C03599=1028.840,190.655,-111.620,169.303,45.603,158.612
C03600=1028.846,190.904,-111.645,169.306,45.600,158.612
C03601=1028.852,191.152,-111.668,169.310,45.598,158.612
C03602=1028.858,191.400,-111.692,169.315,45.595,158.612
C03603=1028.864,191.650,-111.717,169.318,45.592,158.612
C03604=1028.870,191.898,-111.740,169.321,45.590,158.612
C03605=1028.876,192.147,-111.765,169.325,45.587,158.612
C03606=1028.881,192.396,-111.788,169.328,45.585,158.611
C03607=1028.887,192.645,-111.812,169.332,45.583,158.611
C03608=1028.893,192.894,-111.836,169.335,45.580,158.611
C03609=1028.899,193.142,-111.860,169.338,45.578,158.611
C03610=1028.905,193.391,-111.884,169.343,45.575,158.611
C03611=1028.911,193.640,-111.908,169.346,45.572,158.611
C03612=1028.917,193.889,-111.933,169.350,45.570,158.611
C03613=1028.923,194.137,-111.956,169.353,45.567,158.610
C03614=1028.929,194.386,-111.981,169.357,45.565,158.610
C03615=1028.935,194.635,-112.005,169.360,45.563,158.610
C03616=1028.941,194.884,-112.029,169.364,45.560,158.610
C03617=1028.947,195.132,-112.053,169.368,45.557,158.610
C03618=1028.953,195.382,-112.078,169.372,45.555,158.610
C03619=1028.959,195.630,-112.101,169.375,45.552,158.610
C03620=1028.966,195.879,-112.125,169.378,45.550,158.610
C03621=1028.971,196.127,-112.149,169.383,45.547,158.609
C03622=1028.978,196.376,-112.173,169.386,45.545,158.609
C03623=1028.983,196.625,-112.198,169.390,45.542,158.609
C03624=1028.990,196.874,-112.222,169.393,45.540,158.609
C03625=1028.995,197.123,-112.246,169.396,45.537,158.609
C03626=1029.002,197.372,-112.270,169.401,45.535,158.609
C03627=1029.007,197.619,-112.295,169.404,45.532,158.609
C03628=1029.014,197.868,-112.319,169.408,45.530,158.609
C03629=1029.019,198.117,-112.343,169.411,45.528,158.609
C03630=1029.026,198.366,-112.367,169.416,45.525,158.609
C03631=1029.032,198.615,-112.392,169.419,45.522,158.608
C03632=1029.038,198.864,-112.416,169.423,45.520,158.608
C03633=1029.044,199.113,-112.440,169.426,45.518,158.608
C03634=1029.050,199.361,-112.465,169.431,45.515,158.608
C03635=1029.057,199.610,-112.489,169.434,45.512,158.608
C03636=1029.062,199.859,-112.513,169.438,45.510,158.608
C03637=1029.068,200.107,-112.537,169.441,45.507,158.608
C03638=1029.074,200.356,-112.562,169.445,45.505,158.608
C03639=1029.081,200.605,-112.587,169.449,45.503,158.607
C03640=1029.086,200.854,-112.611,169.452,45.500,158.607
C03641=1029.092,201.102,-112.636,169.456,45.498,158.607
C03642=1029.098,201.351,-112.660,169.460,45.496,158.607
C03643=1029.104,201.600,-112.685,169.464,45.494,158.607
C03644=1029.110,201.849,-112.710,169.468,45.491,158.607
C03645=1029.116,202.097,-112.734,169.471,45.488,158.607
C03646=1029.122,202.346,-112.760,169.474,45.486,158.607
C03647=1029.128,202.595,-112.784,169.479,45.484,158.607
C03648=1029.134,202.843,-112.809,169.482,45.482,158.607
C03649=1029.140,203.092,-112.833,169.486,45.479,158.607
C03650=1029.146,203.341,-112.858,169.490,45.477,158.606
C03651=1029.151,203.589,-112.883,169.494,45.475,158.606
C03652=1029.157,203.839,-112.908,169.498,45.472,158.606
C03653=1029.182,204.885,-113.012,169.864,45.576,158.667
C03654=1029.194,205.258,-113.051,169.867,45.574,158.667
C03655=1029.203,205.632,-113.091,169.872,45.571,158.667
C03656=1029.213,206.005,-113.130,169.876,45.569,158.667
C03657=1029.223,206.378,-113.169,169.880,45.566,158.667
C03658=1029.230,206.628,-113.195,169.883,45.565,158.667
C03659=1029.236,206.876,-113.221,169.886,45.564,158.667
C03660=1029.243,207.124,-113.248,169.889,45.562,158.667
C03661=1029.250,207.372,-113.274,169.892,45.560,158.667
C03662=1029.256,207.621,-113.301,169.895,45.559,158.667
C03663=1029.263,207.870,-113.327,169.897,45.557,158.667
C03664=1029.270,208.118,-113.353,169.900,45.556,158.667
C03665=1029.277,208.367,-113.380,169.903,45.554,158.667
C03666=1029.284,208.615,-113.406,169.905,45.553,158.667
C03667=1029.290,208.864,-113.433,169.908,45.551,158.667
C03668=1029.297,209.112,-113.459,169.911,45.550,158.667
C03669=1029.304,209.361,-113.485,169.914,45.549,158.667
C03670=1029.309,209.609,-113.512,169.916,45.547,158.666
C03671=1029.317,209.858,-113.538,169.919,45.545,158.666
C03672=1029.324,210.107,-113.565,169.923,45.544,158.666
C03673=1029.330,210.355,-113.591,169.926,45.542,158.666
C03674=1029.337,210.604,-113.618,169.928,45.541,158.667
C03675=1029.343,210.852,-113.644,169.931,45.540,158.667
C03676=1029.350,211.101,-113.670,169.934,45.538,158.666
C03677=1029.356,211.349,-113.697,169.936,45.536,158.666
C03678=1029.363,211.598,-113.723,169.939,45.535,158.666
C03679=1029.370,211.846,-113.751,169.942,45.534,158.666
C03680=1029.376,212.094,-113.777,169.945,45.532,158.666
C03681=1029.383,212.343,-113.804,169.948,45.531,158.666
C03682=1029.389,212.591,-113.830,169.950,45.530,158.666
C03683=1029.396,212.840,-113.856,169.954,45.528,158.666
C03684=1029.403,213.089,-113.883,169.957,45.527,158.667
C03685=1029.409,213.337,-113.910,169.960,45.525,158.667
C03686=1029.416,213.586,-113.937,169.962,45.524,158.667
C03687=1029.422,213.834,-113.963,169.965,45.523,158.667
C03688=1029.429,214.083,-113.990,169.968,45.521,158.667
C03689=1029.436,214.331,-114.017,169.970,45.519,158.666
C03690=1029.442,214.579,-114.044,169.973,45.518,158.666
C03691=1029.449,214.828,-114.071,169.976,45.517,158.666
C03692=1029.456,215.077,-114.097,169.979,45.515,158.666
C03693=1029.462,215.325,-114.124,169.983,45.514,158.666
C03694=1029.469,215.573,-114.151,169.985,45.512,158.666
C03695=1029.476,215.822,-114.178,169.988,45.511,158.667
C03696=1029.482,216.070,-114.204,169.991,45.510,158.667
C03697=1029.489,216.319,-114.232,169.994,45.508,158.667
C03698=1029.496,216.568,-114.258,169.996,45.507,158.667
C03699=1029.502,216.816,-114.285,169.999,45.506,158.667
C03700=1029.509,217.064,-114.312,170.002,45.504,158.667
C03701=1029.516,217.313,-114.339,170.006,45.503,158.667
C03702=1029.523,217.562,-114.365,170.009,45.501,158.667
C03703=1029.529,217.810,-114.393,170.011,45.500,158.667
C03704=1029.536,218.058,-114.419,170.014,45.499,158.667
C03705=1029.543,218.307,-114.447,170.017,45.497,158.667
C03706=1029.549,218.555,-114.473,170.020,45.496,158.667
C03707=1029.556,218.804,-114.499,170.023,45.495,158.667
C03708=1029.563,219.052,-114.527,170.026,45.493,158.667
C03709=1029.570,219.301,-114.553,170.029,45.492,158.667
C03710=1029.579,219.679,-114.594,170.034,45.490,158.667
C03711=1029.589,220.058,-114.636,170.037,45.488,158.667
C03712=1029.599,220.437,-114.678,170.042,45.486,158.667
C03713=1029.609,220.816,-114.719,170.047,45.484,158.667
C03714=1029.616,221.065,-114.746,170.050,45.483,158.667
C03715=1029.623,221.313,-114.773,170.052,45.482,158.667
C03716=1029.630,221.562,-114.800,170.055,45.480,158.667
C03717=1029.636,221.810,-114.828,170.058,45.479,158.667
C03718=1029.642,222.059,-114.855,170.062,45.477,158.667
C03719=1029.649,222.307,-114.882,170.064,45.476,158.667
C03720=1029.656,222.556,-114.910,170.068,45.475,158.667
C03721=1029.662,222.804,-114.936,170.070,45.474,158.667
C03722=1029.669,223.053,-114.964,170.073,45.473,158.667
C03723=1029.676,223.301,-114.991,170.076,45.471,158.667
C03724=1029.682,223.550,-115.018,170.079,45.470,158.667
C03725=1029.689,223.798,-115.046,170.082,45.468,158.667
C03726=1029.695,224.046,-115.073,170.085,45.467,158.667
C03727=1029.701,224.295,-115.100,170.088,45.466,158.668
C03728=1029.709,224.543,-115.127,170.091,45.465,158.668
C03729=1029.716,224.792,-115.155,170.094,45.464,158.668
C03730=1029.722,225.041,-115.182,170.098,45.462,158.668
C03731=1029.729,225.289,-115.210,170.100,45.461,158.668
C03732=1029.735,225.537,-115.237,170.103,45.460,158.668
C03733=1029.742,225.785,-115.264,170.106,45.459,158.668
C03734=1029.749,226.034,-115.291,170.109,45.457,158.668
C03735=1029.755,226.282,-115.319,170.112,45.456,158.668
C03736=1029.763,226.531,-115.346,170.115,45.454,158.668
C03737=1029.769,226.779,-115.374,170.118,45.454,158.668
C03738=1029.776,227.027,-115.402,170.121,45.452,158.668
C03739=1029.782,227.276,-115.428,170.124,45.451,158.668
C03740=1029.789,227.524,-115.455,170.127,45.450,158.668
C03741=1029.796,227.772,-115.483,170.131,45.448,158.668
C03742=1029.803,228.021,-115.511,170.134,45.447,158.668
C03743=1029.809,228.269,-115.539,170.136,45.446,158.668
C03744=1029.816,228.518,-115.566,170.139,45.445,158.668
C03745=1029.823,228.766,-115.594,170.142,45.444,158.669
C03746=1029.829,229.015,-115.622,170.146,45.443,158.669
C03747=1029.835,229.262,-115.649,170.149,45.441,158.669
C03748=1029.842,229.511,-115.676,170.152,45.440,158.669
C03749=1029.848,229.760,-115.704,170.155,45.439,158.669
C03750=1029.855,230.008,-115.732,170.157,45.438,158.669
C03751=1029.862,230.257,-115.759,170.161,45.437,158.669
C03752=1029.868,230.505,-115.787,170.164,45.436,158.669
C03753=1029.875,230.754,-115.815,170.167,45.434,158.669
C03754=1029.882,231.002,-115.843,170.170,45.433,158.669
C03755=1029.888,231.250,-115.870,170.173,45.432,158.669
C03756=1029.895,231.499,-115.899,170.176,45.431,158.669
C03757=1029.901,231.747,-115.927,170.180,45.430,158.669
C03758=1029.908,231.995,-115.955,170.182,45.429,158.669
C03759=1029.914,232.243,-115.982,170.185,45.428,158.670
C03760=1029.921,232.492,-116.010,170.188,45.427,158.670
C03761=1029.928,232.740,-116.038,170.191,45.426,158.670
C03762=1029.933,232.989,-116.066,170.195,45.424,158.670
C03763=1029.940,233.237,-116.094,170.198,45.424,158.670
C03764=1029.947,233.485,-116.122,170.201,45.422,158.670
C03765=1029.954,233.734,-116.150,170.204,45.422,158.670
C03766=1029.964,234.105,-116.192,170.209,45.420,158.670
C03767=1029.973,234.476,-116.234,170.213,45.418,158.670
C03768=1029.984,234.848,-116.275,170.218,45.416,158.671
C03769=1029.994,235.219,-116.317,170.223,45.414,158.671
C03770=1030.000,235.467,-116.345,170.226,45.414,158.671
C03771=1030.006,235.716,-116.373,170.229,45.412,158.671
C03772=1030.013,235.964,-116.401,170.232,45.412,158.671
C03773=1030.020,236.212,-116.429,170.236,45.410,158.671
C03774=1030.026,236.460,-116.457,170.239,45.409,158.671
C03775=1030.033,236.709,-116.485,170.241,45.408,158.671
C03776=1030.040,236.958,-116.513,170.244,45.407,158.671
C03777=1030.047,237.206,-116.542,170.248,45.406,158.671
C03778=1030.053,237.455,-116.570,170.251,45.405,158.672
C03779=1030.060,237.703,-116.597,170.254,45.404,158.672
C03780=1030.067,237.951,-116.626,170.257,45.403,158.672
C03781=1030.073,238.200,-116.654,170.261,45.401,158.672
C03782=1030.080,238.448,-116.682,170.264,45.401,158.672
C03783=1030.087,238.696,-116.710,170.267,45.400,158.672
C03784=1030.093,238.944,-116.738,170.270,45.399,158.672
C03785=1030.100,239.192,-116.767,170.274,45.398,158.672
C03786=1030.106,239.441,-116.795,170.277,45.396,158.672
C03787=1030.113,239.689,-116.823,170.280,45.396,158.673
C03788=1030.120,239.937,-116.851,170.282,45.394,158.673
C03789=1030.126,240.187,-116.880,170.286,45.394,158.673
C03790=1030.133,240.434,-116.908,170.289,45.393,158.673
C03791=1030.139,240.683,-116.936,170.292,45.392,158.673
C03792=1030.146,240.931,-116.965,170.295,45.391,158.673
C03793=1030.153,241.179,-116.993,170.299,45.390,158.673
C03794=1030.159,241.428,-117.022,170.302,45.389,158.673
C03795=1030.166,241.675,-117.050,170.305,45.388,158.674
C03796=1030.172,241.924,-117.078,170.309,45.387,158.674
C03797=1030.179,242.172,-117.107,170.312,45.386,158.674
C03798=1030.186,242.421,-117.136,170.315,45.385,158.674
C03799=1030.193,242.669,-117.164,170.318,45.384,158.674
C03800=1030.199,242.917,-117.193,170.322,45.383,158.674
C03801=1030.206,243.165,-117.222,170.325,45.382,158.674
C03802=1030.212,243.414,-117.250,170.328,45.381,158.675
C03803=1030.219,243.662,-117.278,170.331,45.381,158.675
C03804=1030.225,243.910,-117.307,170.335,45.380,158.675
C03805=1030.232,244.159,-117.335,170.338,45.378,158.675
C03806=1030.239,244.407,-117.364,170.341,45.378,158.675
C03807=1030.245,244.655,-117.394,170.345,45.377,158.675
C03808=1030.251,244.903,-117.423,170.348,45.376,158.675
C03809=1030.258,245.152,-117.450,170.351,45.375,158.676
C03810=1030.264,245.400,-117.479,170.354,45.375,158.676
C03811=1030.270,245.648,-117.508,170.358,45.373,158.676
C03812=1030.277,245.897,-117.538,170.361,45.372,158.676
C03813=1030.284,246.145,-117.566,170.364,45.372,158.676
C03814=1030.290,246.393,-117.595,170.367,45.371,158.676
C03815=1030.297,246.641,-117.624,170.371,45.370,158.677
C03816=1030.303,246.890,-117.653,170.374,45.369,158.677
C03817=1030.310,247.138,-117.681,170.377,45.369,158.677
C03818=1030.317,247.386,-117.710,170.380,45.368,158.677
C03819=1030.323,247.635,-117.740,170.384,45.367,158.677
C03820=1030.329,247.883,-117.769,170.387,45.366,158.677
C03821=1030.335,248.131,-117.798,170.390,45.365,158.678
C03822=1030.346,248.497,-117.840,170.395,45.364,158.678
C03823=1030.355,248.861,-117.883,170.400,45.363,158.678
C03824=1030.365,249.227,-117.926,170.405,45.362,158.678
C03825=1030.374,249.592,-117.968,170.410,45.360,158.679
C03826=1030.381,249.840,-117.997,170.413,45.360,158.679
C03827=1030.387,250.089,-118.027,170.416,45.359,158.679
C03828=1030.394,250.337,-118.055,170.420,45.358,158.679
C03829=1030.401,250.585,-118.084,170.423,45.357,158.679
C03830=1030.407,250.834,-118.113,170.426,45.357,158.680
C03831=1030.414,251.082,-118.142,170.430,45.356,158.680
C03832=1030.420,251.330,-118.172,170.433,45.355,158.680
C03833=1030.427,251.577,-118.201,170.436,45.354,158.680
C03834=1030.434,251.826,-118.230,170.440,45.353,158.680
C03835=1030.440,252.074,-118.259,170.443,45.353,158.680
C03836=1030.447,252.323,-118.288,170.446,45.352,158.681
C03837=1030.453,252.571,-118.318,170.451,45.351,158.681
C03838=1030.460,252.819,-118.346,170.454,45.350,158.681
C03839=1030.467,253.067,-118.375,170.457,45.349,158.681
C03840=1030.474,253.316,-118.405,170.461,45.349,158.681
C03841=1030.480,253.564,-118.434,170.464,45.348,158.682
C03842=1030.487,253.813,-118.464,170.468,45.347,158.682
C03843=1030.494,254.060,-118.492,170.471,45.347,158.682
C03844=1030.500,254.308,-118.521,170.474,45.346,158.682
C03845=1030.507,254.557,-118.551,170.478,45.345,158.682
C03846=1030.514,254.805,-118.580,170.481,45.344,158.682
C03847=1030.520,255.054,-118.610,170.485,45.343,158.683
C03848=1030.527,255.301,-118.638,170.488,45.343,158.683
C03849=1030.534,255.549,-118.668,170.491,45.342,158.683
C03850=1030.541,255.798,-118.697,170.495,45.341,158.683
C03851=1030.547,256.046,-118.726,170.498,45.340,158.683
C03852=1030.554,256.294,-118.756,170.502,45.339,158.684
C03853=1030.560,256.542,-118.785,170.505,45.339,158.684
C03854=1030.568,256.791,-118.814,170.508,45.338,158.684
C03855=1030.575,257.038,-118.844,170.512,45.337,158.684
C03856=1030.581,257.287,-118.873,170.515,45.336,158.684
C03857=1030.588,257.535,-118.903,170.519,45.335,158.685
C03858=1030.594,257.783,-118.932,170.522,45.335,158.685
C03859=1030.602,258.031,-118.961,170.525,45.334,158.685
C03860=1030.608,258.279,-118.990,170.529,45.333,158.685
C03861=1030.615,258.528,-119.020,170.533,45.333,158.685
C03862=1030.622,258.776,-119.049,170.537,45.332,158.686
C03863=1030.629,259.024,-119.079,170.540,45.331,158.686
C03864=1030.636,259.273,-119.109,170.544,45.331,158.686
C03865=1030.643,259.520,-119.138,170.547,45.330,158.686
C03866=1030.650,259.769,-119.167,170.551,45.329,158.686
C03867=1030.656,260.017,-119.196,170.554,45.328,158.687
C03868=1030.663,260.265,-119.227,170.558,45.327,158.687
C03869=1030.669,260.513,-119.256,170.561,45.327,158.687
C03870=1030.676,260.762,-119.286,170.564,45.327,158.687
C03871=1030.684,261.009,-119.315,170.568,45.326,158.688
C03872=1030.691,261.258,-119.344,170.571,45.325,158.688
C03873=1030.696,261.505,-119.375,170.575,45.324,158.688
C03874=1030.703,261.754,-119.404,170.579,45.324,158.688
C03875=1030.710,262.002,-119.434,170.583,45.323,158.688
C03876=1030.717,262.250,-119.464,170.586,45.322,158.689
C03877=1030.724,262.497,-119.494,170.589,45.322,158.689
C03878=1030.733,262.862,-119.538,170.594,45.321,158.689
C03879=1030.743,263.226,-119.582,170.600,45.320,158.690
C03880=1030.752,263.590,-119.626,170.606,45.319,158.690
C03881=1030.762,263.954,-119.670,170.611,45.319,158.690
C03882=1030.769,264.202,-119.700,170.614,45.318,158.691
C03883=1030.775,264.450,-119.729,170.618,45.317,158.691
C03884=1030.783,264.698,-119.759,170.621,45.317,158.691
C03885=1030.789,264.947,-119.790,170.624,45.316,158.691
C03886=1030.796,265.194,-119.819,170.629,45.316,158.692
C03887=1030.803,265.442,-119.850,170.632,45.315,158.692
C03888=1030.809,265.690,-119.879,170.636,45.314,158.692
C03889=1030.816,265.938,-119.910,170.639,45.314,158.692
C03890=1030.823,266.187,-119.939,170.643,45.313,158.693
C03891=1030.829,266.435,-119.969,170.646,45.313,158.693
C03892=1030.836,266.683,-119.999,170.650,45.312,158.693
C03893=1030.843,266.932,-120.030,170.654,45.312,158.694
C03894=1030.849,267.179,-120.060,170.658,45.311,158.694
C03895=1030.856,267.427,-120.090,170.661,45.311,158.694
C03896=1030.863,267.676,-120.121,170.665,45.310,158.694
C03897=1030.869,267.923,-120.150,170.668,45.310,158.695
C03898=1030.876,268.172,-120.181,170.672,45.309,158.695
C03899=1030.883,268.420,-120.211,170.676,45.309,158.695
C03900=1030.890,268.667,-120.242,170.680,45.308,158.695
C03901=1030.896,268.915,-120.272,170.683,45.308,158.696
C03902=1030.903,269.164,-120.302,170.687,45.307,158.696
C03903=1030.909,269.411,-120.333,170.690,45.307,158.696
C03904=1030.916,269.660,-120.363,170.694,45.306,158.696
C03905=1030.924,269.908,-120.393,170.698,45.306,158.697
C03906=1030.929,270.156,-120.423,170.702,45.306,158.697
C03907=1030.937,270.404,-120.454,170.705,45.305,158.697
C03908=1030.943,270.652,-120.485,170.709,45.305,158.698
C03909=1030.950,270.900,-120.515,170.712,45.304,158.698
C03910=1030.956,271.148,-120.545,170.717,45.304,158.698
C03911=1030.963,271.396,-120.576,170.720,45.304,158.699
C03912=1030.970,271.644,-120.607,170.724,45.303,158.699
C03913=1030.977,271.892,-120.637,170.727,45.303,158.699
C03914=1030.983,272.140,-120.667,170.732,45.303,158.700
C03915=1030.989,272.389,-120.698,170.735,45.302,158.700
C03916=1030.997,272.636,-120.729,170.739,45.302,158.700
C03917=1031.003,272.885,-120.760,170.742,45.302,158.700
C03918=1031.010,273.132,-120.790,170.746,45.301,158.701
C03919=1031.017,273.380,-120.821,170.750,45.301,158.701
C03920=1031.024,273.628,-120.851,170.754,45.300,158.701
C03921=1031.031,273.876,-120.882,170.757,45.300,158.702
C03922=1031.036,274.124,-120.913,170.761,45.300,158.702
C03923=1031.043,274.372,-120.943,170.764,45.299,158.702
C03924=1031.050,274.620,-120.974,170.769,45.299,158.703
C03925=1031.057,274.869,-121.005,170.772,45.299,158.703
C03926=1031.064,275.116,-121.036,170.776,45.298,158.703
C03927=1031.071,275.365,-121.067,170.780,45.298,158.704
C03928=1031.077,275.612,-121.098,170.784,45.298,158.704
C03929=1031.084,275.860,-121.128,170.788,45.298,158.704
C03930=1031.091,276.108,-121.159,170.791,45.297,158.705
C03931=1031.097,276.357,-121.190,170.795,45.297,158.705
C03932=1031.104,276.604,-121.221,170.799,45.296,158.705
C03933=1031.111,276.853,-121.252,170.803,45.296,158.705
C03934=1031.121,277.221,-121.298,170.808,45.296,158.706
C03935=1031.131,277.589,-121.343,170.815,45.295,158.706
C03936=1031.141,277.957,-121.390,170.820,45.295,158.707
C03937=1031.151,278.327,-121.436,170.826,45.294,158.707
C03938=1031.157,278.574,-121.467,170.830,45.294,158.708
C03939=1031.164,278.822,-121.498,170.833,45.294,158.708
C03940=1031.171,279.070,-121.529,170.837,45.294,158.709
C03941=1031.177,279.319,-121.560,170.841,45.294,158.709
C03942=1031.184,279.566,-121.592,170.845,45.293,158.709
C03943=1031.191,279.814,-121.623,170.849,45.293,158.710
C03944=1031.197,280.062,-121.654,170.853,45.293,158.710
C03945=1031.204,280.310,-121.686,170.857,45.293,158.710
C03946=1031.211,280.559,-121.717,170.860,45.293,158.711
C03947=1031.218,280.806,-121.747,170.865,45.292,158.711
C03948=1031.225,281.054,-121.779,170.869,45.292,158.711
C03949=1031.232,281.302,-121.810,170.872,45.292,158.712
C03950=1031.238,281.550,-121.842,170.876,45.292,158.712
C03951=1031.245,281.798,-121.873,170.880,45.292,158.712
C03952=1031.252,282.046,-121.905,170.884,45.291,158.713
C03953=1031.258,282.294,-121.936,170.888,45.291,158.713
C03954=1031.265,282.542,-121.968,170.892,45.291,158.714
C03955=1031.272,282.790,-121.998,170.896,45.291,158.714
C03956=1031.278,283.038,-122.030,170.900,45.290,158.714
C03957=1031.285,283.286,-122.061,170.904,45.290,158.715
C03958=1031.292,283.534,-122.093,170.908,45.290,158.715
C03959=1031.299,283.781,-122.123,170.912,45.290,158.716
C03960=1031.306,284.029,-122.155,170.916,45.290,158.716
C03961=1031.313,284.277,-122.186,170.920,45.290,158.716
C03962=1031.319,284.525,-122.218,170.923,45.290,158.717
C03963=1031.326,284.772,-122.250,170.928,45.290,158.717
C03964=1031.333,285.020,-122.281,170.932,45.289,158.717
C03965=1031.340,285.268,-122.313,170.935,45.289,158.718
C03966=1031.347,285.516,-122.344,170.940,45.289,158.718
C03967=1031.353,285.764,-122.376,170.944,45.289,158.719
C03968=1031.360,286.012,-122.407,170.948,45.289,158.719
C03969=1031.367,286.260,-122.438,170.952,45.289,158.719
C03970=1031.374,286.508,-122.470,170.956,45.289,158.720
C03971=1031.381,286.756,-122.502,170.960,45.288,158.720
C03972=1031.388,287.004,-122.534,170.964,45.289,158.721
C03973=1031.395,287.251,-122.565,170.968,45.289,158.721
C03974=1031.401,287.500,-122.597,170.972,45.288,158.721
C03975=1031.408,287.747,-122.629,170.976,45.289,158.722
C03976=1031.414,287.995,-122.661,170.980,45.289,158.722
C03977=1031.421,288.243,-122.692,170.985,45.288,158.723
C03978=1031.429,288.491,-122.725,170.988,45.288,158.723
C03979=1031.435,288.739,-122.756,170.992,45.289,158.723
C03980=1031.442,288.987,-122.788,170.997,45.288,158.724
C03981=1031.448,289.234,-122.820,171.000,45.288,158.724
C03982=1031.455,289.482,-122.852,171.005,45.288,158.725
C03983=1031.462,289.729,-122.884,171.009,45.288,158.725
C03984=1031.469,289.978,-122.916,171.013,45.289,158.726
C03985=1031.476,290.226,-122.948,171.017,45.288,158.726
C03986=1031.482,290.473,-122.980,171.021,45.288,158.726
C03987=1031.489,290.721,-123.011,171.026,45.288,158.727
C03988=1031.496,290.969,-123.044,171.029,45.288,158.727
C03989=1031.503,291.218,-123.076,171.034,45.289,158.728
C03990=1031.514,291.598,-123.125,171.040,45.289,158.728
C03991=1031.524,291.978,-123.174,171.047,45.288,158.729
C03992=1031.535,292.359,-123.224,171.052,45.289,158.730
C03993=1031.546,292.739,-123.273,171.059,45.288,158.730
C03994=1031.552,292.987,-123.305,171.063,45.289,158.731
C03995=1031.559,293.236,-123.337,171.067,45.289,158.731
C03996=1031.566,293.483,-123.370,171.071,45.289,158.732
C03997=1031.573,293.731,-123.402,171.076,45.289,158.732
C03998=1031.579,293.978,-123.434,171.080,45.289,158.733
C03999=1031.586,294.227,-123.467,171.084,45.290,158.733
C04000=1031.593,294.474,-123.499,171.088,45.289,158.734
C04001=1031.599,294.722,-123.532,171.093,45.290,158.734
C04002=1031.606,294.969,-123.563,171.097,45.290,158.735
C04003=1031.613,295.218,-123.596,171.100,45.290,158.735
C04004=1031.619,295.465,-123.629,171.105,45.290,158.735
C04005=1031.626,295.713,-123.661,171.110,45.290,158.736
C04006=1031.633,295.961,-123.694,171.114,45.290,158.736
C04007=1031.640,296.209,-123.727,171.117,45.291,158.737
C04008=1031.647,296.456,-123.759,171.122,45.291,158.737
C04009=1031.653,296.703,-123.792,171.127,45.291,158.738
C04010=1031.660,296.952,-123.825,171.131,45.292,158.739
C04011=1031.667,297.199,-123.857,171.134,45.292,158.739
C04012=1031.673,297.447,-123.890,171.139,45.292,158.739
C04013=1031.680,297.695,-123.923,171.144,45.292,158.740
C04014=1031.686,297.942,-123.956,171.148,45.293,158.741
C04015=1031.694,298.190,-123.988,171.151,45.292,158.741
C04016=1031.700,298.438,-124.021,171.156,45.293,158.741
C04017=1031.707,298.686,-124.054,171.161,45.293,158.742
C04018=1031.714,298.934,-124.086,171.165,45.293,158.742
C04019=1031.721,299.181,-124.120,171.170,45.294,158.743
C04020=1031.728,299.429,-124.153,171.173,45.294,158.744
C04021=1031.734,299.676,-124.185,171.178,45.294,158.744
C04022=1031.741,299.924,-124.218,171.182,45.294,158.744
C04023=1031.748,300.172,-124.251,171.187,45.295,158.745
C04024=1031.754,300.420,-124.283,171.191,45.295,158.746
C04025=1031.762,300.667,-124.317,171.196,45.295,158.746
C04026=1031.768,300.915,-124.349,171.199,45.296,158.747
C04027=1031.775,301.163,-124.383,171.204,45.296,158.747
C04028=1031.782,301.411,-124.415,171.209,45.296,158.748
C04029=1031.790,301.658,-124.448,171.213,45.297,158.748
C04030=1031.796,301.905,-124.481,171.218,45.297,158.749
C04031=1031.803,302.154,-124.514,171.222,45.297,158.749
C04032=1031.810,302.400,-124.547,171.226,45.298,158.750
C04033=1031.817,302.649,-124.580,171.230,45.298,158.750
C04034=1031.823,302.896,-124.613,171.235,45.298,158.751
C04035=1031.830,303.144,-124.647,171.239,45.298,158.751
C04036=1031.837,303.391,-124.679,171.244,45.298,158.752
C04037=1031.844,303.640,-124.712,171.248,45.299,158.752
C04038=1031.851,303.887,-124.746,171.253,45.299,158.753
C04039=1031.858,304.135,-124.779,171.258,45.299,158.753
C04040=1031.866,304.382,-124.812,171.261,45.300,158.754
C04041=1031.872,304.630,-124.845,171.266,45.300,158.755
C04042=1031.879,304.877,-124.879,171.270,45.301,158.755
C04043=1031.886,305.125,-124.911,171.275,45.302,158.756
C04044=1031.894,305.372,-124.944,171.280,45.302,158.756
C04045=1031.900,305.621,-124.978,171.284,45.302,158.757
C04046=1031.911,306.018,-125.031,171.291,45.303,158.758
C04047=1031.922,306.416,-125.084,171.299,45.303,158.759
C04048=1031.934,306.814,-125.137,171.306,45.304,158.760
C04049=1031.945,307.211,-125.191,171.313,45.304,158.760
C04050=1031.952,307.459,-125.224,171.317,45.305,158.761
C04051=1031.960,307.706,-125.258,171.322,45.306,158.762
C04052=1031.967,307.953,-125.291,171.327,45.306,158.762
C04053=1031.974,308.202,-125.324,171.331,45.306,158.763
C04054=1031.981,308.449,-125.358,171.336,45.307,158.763
C04055=1031.989,308.697,-125.391,171.341,45.307,158.764
C04056=1031.995,308.944,-125.424,171.345,45.307,158.764
C04057=1032.002,309.192,-125.458,171.350,45.308,158.765
C04058=1032.010,309.440,-125.492,171.355,45.308,158.766
C04059=1032.017,309.687,-125.526,171.359,45.309,158.766
C04060=1032.024,309.935,-125.558,171.364,45.309,158.767
C04061=1032.031,310.182,-125.591,171.368,45.310,158.767
C04062=1032.038,310.430,-125.625,171.373,45.310,158.768
C04063=1032.045,310.678,-125.659,171.378,45.311,158.769
C04064=1032.053,310.925,-125.692,171.382,45.311,158.769
C04065=1032.060,311.173,-125.725,171.387,45.312,158.770
C04066=1032.067,311.421,-125.759,171.392,45.312,158.770
C04067=1032.074,311.668,-125.794,171.396,45.312,158.771
C04068=1032.081,311.915,-125.828,171.401,45.313,158.772
C04069=1032.088,312.163,-125.862,171.406,45.314,158.772
C04070=1032.094,312.411,-125.896,171.410,45.315,158.773
C04071=1032.101,312.658,-125.930,171.415,45.315,158.774
C04072=1032.108,312.906,-125.963,171.420,45.316,158.774
C04073=1032.115,313.154,-125.998,171.425,45.317,158.775
C04074=1032.122,313.401,-126.032,171.429,45.317,158.775
C04075=1032.129,313.648,-126.066,171.434,45.318,158.776
C04076=1032.136,313.896,-126.101,171.439,45.319,158.777
C04077=1032.142,314.143,-126.134,171.443,45.319,158.777
C04078=1032.149,314.391,-126.169,171.448,45.320,158.778
C04079=1032.156,314.638,-126.203,171.453,45.321,158.779
C04080=1032.164,314.886,-126.237,171.458,45.321,158.779
C04081=1032.170,315.134,-126.271,171.462,45.322,158.780
C04082=1032.178,315.381,-126.306,171.467,45.323,158.781
C04083=1032.184,315.629,-126.340,171.472,45.323,158.781
C04084=1032.192,315.876,-126.375,171.477,45.324,158.782
C04085=1032.199,316.124,-126.409,171.482,45.325,158.783
C04086=1032.205,316.372,-126.443,171.486,45.325,158.783
C04087=1032.212,316.618,-126.477,171.491,45.326,158.784
C04088=1032.219,316.866,-126.512,171.496,45.327,158.785
C04089=1032.226,317.113,-126.546,171.501,45.328,158.785
C04090=1032.233,317.361,-126.580,171.505,45.329,158.786
C04091=1032.240,317.609,-126.614,171.510,45.329,158.787
C04092=1032.247,317.856,-126.649,171.515,45.330,158.787
C04093=1032.254,318.104,-126.683,171.520,45.331,158.788
C04094=1032.261,318.351,-126.718,171.524,45.332,158.789
C04095=1032.269,318.599,-126.753,171.529,45.332,158.789
C04096=1032.276,318.847,-126.787,171.535,45.333,158.790
C04097=1032.283,319.094,-126.822,171.540,45.334,158.791
C04098=1032.290,319.342,-126.856,171.545,45.335,158.792
C04099=1032.297,319.589,-126.891,171.549,45.336,158.792
C04100=1032.304,319.836,-126.925,171.554,45.336,158.793
C04101=1032.311,320.084,-126.960,171.559,45.337,158.794
C04102=1032.323,320.486,-127.016,171.567,45.339,158.795
C04103=1032.334,320.888,-127.073,171.575,45.340,158.796
C04104=1032.347,321.292,-127.129,171.583,45.342,158.797
C04105=1032.358,321.694,-127.185,171.591,45.342,158.798
C04106=1032.366,321.941,-127.220,171.596,45.343,158.799
C04107=1032.372,322.189,-127.255,171.601,45.344,158.800
C04108=1032.380,322.436,-127.289,171.606,45.345,158.800
C04109=1032.387,322.684,-127.324,171.612,45.346,158.801
C04110=1032.394,322.932,-127.359,171.616,45.347,158.802
C04111=1032.401,323.179,-127.394,171.621,45.348,158.803
C04112=1032.409,323.426,-127.428,171.626,45.349,158.803
C04113=1032.417,323.674,-127.463,171.631,45.349,158.804
C04114=1032.424,323.921,-127.498,171.637,45.350,158.805
C04115=1032.431,324.168,-127.533,171.642,45.351,158.805
C04116=1032.438,324.416,-127.568,171.647,45.353,158.806
C04117=1032.446,324.663,-127.603,171.651,45.353,158.807
C04118=1032.452,324.911,-127.637,171.656,45.354,158.808
C04119=1032.460,325.159,-127.672,171.662,45.355,158.809
C04120=1032.467,325.406,-127.707,171.667,45.356,158.809
C04121=1032.475,325.653,-127.742,171.672,45.357,158.810
C04122=1032.482,325.901,-127.777,171.677,45.358,158.811
C04123=1032.490,326.148,-127.813,171.682,45.358,158.811
C04124=1032.497,326.395,-127.848,171.688,45.360,158.812
C04125=1032.505,326.643,-127.883,171.692,45.361,158.813
C04126=1032.512,326.890,-127.917,171.697,45.362,158.814
C04127=1032.520,327.138,-127.953,171.703,45.362,158.815
C04128=1032.527,327.385,-127.987,171.708,45.363,158.815
C04129=1032.534,327.633,-128.022,171.713,45.365,158.816
C04130=1032.542,327.880,-128.057,171.718,45.366,158.817
C04131=1032.549,328.127,-128.093,171.724,45.366,158.818
C04132=1032.556,328.375,-128.129,171.729,45.368,158.819
C04133=1032.563,328.622,-128.164,171.734,45.369,158.819
C04134=1032.571,328.870,-128.200,171.739,45.370,158.820
C04135=1032.578,329.117,-128.235,171.745,45.371,158.821
C04136=1032.586,329.364,-128.270,171.749,45.372,158.822
C04137=1032.593,329.612,-128.306,171.755,45.373,158.823
C04138=1032.600,329.859,-128.341,171.759,45.374,158.823
C04139=1032.607,330.107,-128.377,171.766,45.375,158.824
C04140=1032.614,330.354,-128.412,171.770,45.376,158.825
C04141=1032.622,330.601,-128.449,171.775,45.378,158.826
C04142=1032.629,330.849,-128.484,171.782,45.379,158.827
C04143=1032.636,331.096,-128.520,171.786,45.380,158.827
C04144=1032.643,331.343,-128.556,171.792,45.382,158.828
C04145=1032.651,331.591,-128.591,171.797,45.382,158.829
C04146=1032.658,331.837,-128.627,171.802,45.384,158.830
C04147=1032.666,332.086,-128.662,171.807,45.385,158.831
C04148=1032.673,332.332,-128.698,171.813,45.386,158.832
C04149=1032.681,332.580,-128.734,171.819,45.387,158.833
C04150=1032.688,332.828,-128.770,171.823,45.388,158.833
C04151=1032.695,333.075,-128.805,171.829,45.389,158.834
C04152=1032.703,333.322,-128.842,171.835,45.391,158.835
C04153=1032.710,333.569,-128.878,171.839,45.392,158.836
C04154=1032.717,333.817,-128.913,171.846,45.393,158.837
C04155=1032.725,334.064,-128.949,171.851,45.395,158.838
C04156=1032.732,334.311,-128.985,171.856,45.396,158.839
C04157=1032.740,334.558,-129.021,171.862,45.397,158.839
C04158=1032.752,334.957,-129.079,171.871,45.399,158.841
C04159=1032.764,335.355,-129.138,171.879,45.401,158.842
C04160=1032.775,335.753,-129.195,171.888,45.403,158.844
C04161=1032.787,336.151,-129.254,171.897,45.405,158.845
C04162=1032.795,336.398,-129.290,171.902,45.407,158.846
C04163=1032.802,336.645,-129.326,171.908,45.408,158.847
C04164=1032.810,336.892,-129.362,171.913,45.410,158.848
C04165=1032.816,337.140,-129.399,171.918,45.411,158.849
C04166=1032.824,337.387,-129.435,171.924,45.412,158.850
C04167=1032.831,337.634,-129.471,171.929,45.414,158.851
C04168=1032.839,337.882,-129.507,171.935,45.415,158.851
C04169=1032.847,338.128,-129.544,171.940,45.417,158.852
C04170=1032.855,338.376,-129.581,171.947,45.418,158.853
C04171=1032.861,338.624,-129.617,171.952,45.419,158.854
C04172=1032.869,338.870,-129.653,171.958,45.421,158.855
C04173=1032.876,339.118,-129.689,171.963,45.422,158.856
C04174=1032.884,339.365,-129.726,171.968,45.424,158.857
C04175=1032.892,339.612,-129.763,171.974,45.425,158.858
C04176=1032.899,339.860,-129.799,171.980,45.427,158.859
C04177=1032.907,340.107,-129.836,171.986,45.428,158.860
C04178=1032.914,340.354,-129.873,171.991,45.430,158.861
C04179=1032.922,340.602,-129.909,171.997,45.431,158.862
C04180=1032.930,340.848,-129.945,172.002,45.432,158.863
C04181=1032.936,341.095,-129.982,172.008,45.434,158.864
C04182=1032.944,341.342,-130.019,172.013,45.436,158.865
C04183=1032.951,341.590,-130.056,172.020,45.437,158.866
C04184=1032.959,341.837,-130.093,172.025,45.439,158.867
C04185=1032.967,342.084,-130.129,172.031,45.440,158.868
C04186=1032.974,342.331,-130.167,172.036,45.442,158.868
C04187=1032.982,342.578,-130.203,172.043,45.444,158.870
C04188=1032.989,342.826,-130.240,172.048,45.445,158.870
C04189=1032.997,343.073,-130.277,172.054,45.446,158.871
C04190=1033.004,343.321,-130.314,172.060,45.448,158.873
C04191=1033.012,343.567,-130.351,172.065,45.450,158.873
C04192=1033.019,343.815,-130.388,172.072,45.451,158.875
C04193=1033.027,344.061,-130.425,172.077,45.453,158.875
C04194=1033.035,344.309,-130.462,172.083,45.455,158.877
C04195=1033.042,344.556,-130.499,172.088,45.456,158.877
C04196=1033.050,344.803,-130.536,172.095,45.458,158.879
C04197=1033.057,345.050,-130.574,172.100,45.460,158.879
C04198=1033.065,345.297,-130.611,172.106,45.461,158.881
C04199=1033.072,345.544,-130.647,172.112,45.463,158.882
C04200=1033.080,345.792,-130.685,172.118,45.465,158.883
C04201=1033.088,346.038,-130.722,172.124,45.466,158.884
C04202=1033.095,346.286,-130.759,172.129,45.468,158.885
C04203=1033.103,346.533,-130.797,172.136,45.470,158.886
C04204=1033.111,346.780,-130.834,172.142,45.471,158.887
C04205=1033.119,347.027,-130.871,172.147,45.473,158.888
C04206=1033.126,347.274,-130.909,172.154,45.475,158.889
C04207=1033.134,347.521,-130.946,172.160,45.477,158.890
C04208=1033.141,347.768,-130.983,172.165,45.478,158.891
C04209=1033.150,348.016,-131.020,172.171,45.480,158.892
C04210=1033.157,348.263,-131.058,172.178,45.482,158.893
C04211=1033.165,348.509,-131.096,172.183,45.484,158.894
C04212=1033.173,348.756,-131.133,172.189,45.485,158.895
C04213=1033.180,349.003,-131.171,172.196,45.487,158.896
C04214=1033.193,349.398,-131.231,172.205,45.490,158.898
C04215=1033.204,349.793,-131.291,172.215,45.493,158.900
C04216=1033.217,350.188,-131.351,172.224,45.496,158.902
C04217=1033.230,350.582,-131.412,172.235,45.499,158.903
C04218=1033.237,350.829,-131.449,172.240,45.501,158.904
C04219=1033.245,351.077,-131.488,172.247,45.503,158.906
C04220=1033.252,351.324,-131.525,172.253,45.505,158.907
C04221=1033.260,351.571,-131.563,172.258,45.507,158.908
C04222=1033.268,351.818,-131.601,172.265,45.509,158.909
C04223=1033.276,352.064,-131.639,172.271,45.511,158.910
C04224=1033.283,352.311,-131.677,172.277,45.512,158.911
C04225=1033.291,352.559,-131.715,172.283,45.514,158.912
C04226=1033.299,352.806,-131.753,172.289,45.516,158.913
C04227=1033.307,353.053,-131.791,172.296,45.519,158.915
C04228=1033.315,353.300,-131.828,172.302,45.520,158.916
C04229=1033.322,353.546,-131.866,172.308,45.522,158.917
C04230=1033.330,353.793,-131.905,172.314,45.524,158.918
C04231=1033.338,354.041,-131.943,172.321,45.526,158.919
C04232=1033.346,354.288,-131.981,172.327,45.529,158.920
C04233=1033.354,354.534,-132.019,172.334,45.530,158.921
C04234=1033.362,354.781,-132.057,172.340,45.532,158.923
C04235=1033.369,355.028,-132.095,172.346,45.535,158.924
C04236=1033.378,355.276,-132.134,172.352,45.537,158.925
C04237=1033.385,355.522,-132.172,172.359,45.538,158.926
C04238=1033.393,355.769,-132.210,172.365,45.541,158.927
C04239=1033.401,356.016,-132.249,172.372,45.543,158.929
C04240=1033.409,356.263,-132.287,172.378,45.545,158.930
C04241=1033.417,356.510,-132.326,172.384,45.547,158.931
C04242=1033.425,356.757,-132.364,172.390,45.549,158.932
C04243=1033.433,357.004,-132.403,172.397,45.551,158.933
C04244=1033.440,357.251,-132.441,172.403,45.554,158.935
C04245=1033.449,357.498,-132.480,172.410,45.555,158.936
C04246=1033.456,357.744,-132.518,172.417,45.558,158.937
C04247=1033.464,357.991,-132.556,172.423,45.560,158.938
C04248=1033.472,358.239,-132.595,172.430,45.562,158.939
C04249=1033.480,358.485,-132.634,172.435,45.564,158.941
C04250=1033.488,358.732,-132.673,172.442,45.566,158.942
C04251=1033.497,358.979,-132.711,172.448,45.569,158.943
C04252=1033.504,359.226,-132.750,172.455,45.571,158.944
C04253=1033.513,359.472,-132.789,172.461,45.573,158.946
C04254=1033.521,359.719,-132.827,172.468,45.575,158.947
C04255=1033.529,359.967,-132.866,172.475,45.578,158.948
C04256=1033.537,360.212,-132.905,172.481,45.580,158.949
C04257=1033.545,360.460,-132.944,172.488,45.582,158.951
C04258=1033.552,360.707,-132.983,172.495,45.584,158.952
C04259=1033.561,360.954,-133.022,172.501,45.587,158.953
C04260=1033.568,361.200,-133.060,172.508,45.589,158.955
C04261=1033.577,361.447,-133.100,172.515,45.591,158.956
C04262=1033.585,361.694,-133.138,172.521,45.594,158.957
C04263=1033.593,361.941,-133.178,172.528,45.596,158.958
C04264=1033.601,362.188,-133.218,172.535,45.599,158.960
C04265=1033.609,362.434,-133.256,172.541,45.601,158.961
C04266=1033.616,362.681,-133.296,172.548,45.603,158.962
C04267=1033.625,362.928,-133.335,172.555,45.606,158.964
C04268=1033.633,363.175,-133.374,172.561,45.608,158.965
C04269=1033.641,363.422,-133.414,172.568,45.610,158.966
C04270=1033.653,363.822,-133.477,172.579,45.615,158.968
C04271=1033.667,364.224,-133.541,172.590,45.619,158.971
C04272=1033.680,364.624,-133.606,172.602,45.622,158.973
C04273=1033.693,365.025,-133.669,172.612,45.626,158.975
C04274=1033.701,365.272,-133.709,172.619,45.629,158.976
C04275=1033.710,365.518,-133.748,172.626,45.632,158.978
C04276=1033.717,365.765,-133.788,172.633,45.634,158.979
C04277=1033.726,366.012,-133.827,172.640,45.637,158.981
C04278=1033.734,366.258,-133.867,172.647,45.639,158.982
C04279=1033.742,366.505,-133.907,172.654,45.641,158.983
C04280=1033.751,366.752,-133.946,172.661,45.644,158.985
C04281=1033.759,366.999,-133.986,172.668,45.647,158.986
C04282=1033.767,367.246,-134.025,172.675,45.650,158.988
C04283=1033.776,367.492,-134.066,172.681,45.652,158.989
C04284=1033.784,367.739,-134.105,172.689,45.654,158.990
C04285=1033.792,367.985,-134.145,172.696,45.657,158.992
C04286=1033.801,368.232,-134.184,172.703,45.659,158.993
C04287=1033.808,368.479,-134.224,172.710,45.662,158.995
C04288=1033.817,368.725,-134.264,172.717,45.665,158.996
C04289=1033.825,368.972,-134.304,172.724,45.667,158.997
C04290=1033.834,369.219,-134.344,172.731,45.670,158.999
C04291=1033.843,369.465,-134.384,172.738,45.673,159.000
C04292=1033.850,369.712,-134.424,172.745,45.676,159.002
C04293=1033.859,369.959,-134.465,172.753,45.678,159.003
C04294=1033.867,370.206,-134.504,172.760,45.681,159.005
C04295=1033.875,370.452,-134.545,172.767,45.684,159.006
C04296=1033.883,370.699,-134.585,172.774,45.687,159.008
C04297=1033.892,370.945,-134.625,172.782,45.689,159.009
C04298=1033.901,371.192,-134.666,172.789,45.692,159.011
C04299=1033.908,371.439,-134.705,172.796,45.695,159.012
C04300=1033.917,371.685,-134.746,172.804,45.698,159.014
C04301=1033.925,371.931,-134.786,172.811,45.701,159.015
C04302=1033.934,372.178,-134.827,172.818,45.704,159.017
C04303=1033.941,372.425,-134.867,172.825,45.707,159.018
C04304=1033.950,372.671,-134.907,172.833,45.709,159.020
C04305=1033.959,372.918,-134.948,172.840,45.712,159.021
C04306=1033.967,373.164,-134.989,172.847,45.715,159.023
C04307=1033.975,373.410,-135.029,172.855,45.718,159.024
C04308=1033.984,373.657,-135.070,172.862,45.721,159.026
C04309=1033.992,373.903,-135.110,172.870,45.724,159.027
C04310=1034.001,374.150,-135.151,172.877,45.727,159.029
C04311=1034.010,374.396,-135.191,172.884,45.730,159.030
C04312=1034.018,374.642,-135.232,172.892,45.733,159.032
C04313=1034.026,374.889,-135.273,172.899,45.735,159.033
C04314=1034.034,375.136,-135.314,172.907,45.739,159.035
C04315=1034.044,375.382,-135.354,172.914,45.742,159.037
C04316=1034.052,375.629,-135.395,172.921,45.745,159.038
C04317=1034.060,375.876,-135.436,172.929,45.748,159.040
C04318=1034.069,376.123,-135.477,172.936,45.751,159.041
C04319=1034.078,376.368,-135.518,172.944,45.753,159.043
C04320=1034.087,376.615,-135.559,172.952,45.757,159.045
C04321=1034.095,376.861,-135.599,172.959,45.759,159.046
C04322=1034.103,377.108,-135.640,172.967,45.763,159.048
C04323=1034.112,377.354,-135.681,172.975,45.766,159.049
C04324=1034.121,377.601,-135.722,172.982,45.769,159.051
C04325=1034.130,377.848,-135.763,172.990,45.772,159.053
C04326=1034.137,378.058,-135.799,172.997,45.775,159.054
C04327=1034.145,378.269,-135.834,173.003,45.777,159.055
C04328=1034.152,378.480,-135.869,173.010,45.780,159.057
C04329=1034.159,378.690,-135.904,173.016,45.782,159.058
C04330=1034.166,378.901,-135.940,173.023,45.785,159.060
C04331=1034.174,379.112,-135.975,173.029,45.788,159.061
C04332=1034.181,379.323,-136.010,173.036,45.791,159.062
C04333=1034.189,379.533,-136.046,173.043,45.794,159.064
C04334=1034.197,379.780,-136.087,173.050,45.797,159.066
C04335=1034.205,380.026,-136.129,173.059,45.800,159.067
C04336=1034.214,380.273,-136.171,173.067,45.804,159.069
C04337=1034.223,380.519,-136.212,173.074,45.807,159.071
C04338=1034.231,380.766,-136.253,173.083,45.810,159.073
C04339=1034.240,381.012,-136.295,173.090,45.814,159.074
C04340=1034.249,381.258,-136.337,173.098,45.817,159.076
C04341=1034.258,381.504,-136.378,173.106,45.820,159.078
C04342=1034.267,381.751,-136.420,173.114,45.824,159.079
C04343=1034.275,381.997,-136.462,173.122,45.827,159.081
C04344=1034.284,382.243,-136.503,173.130,45.830,159.083
C04345=1034.293,382.490,-136.545,173.139,45.833,159.085
C04346=1034.301,382.736,-136.587,173.146,45.837,159.086
C04347=1034.310,382.982,-136.629,173.154,45.840,159.088
C04348=1034.319,383.229,-136.670,173.162,45.843,159.090
C04349=1034.328,383.474,-136.713,173.170,45.847,159.092
C04350=1034.337,383.721,-136.755,173.178,45.850,159.093
C04351=1034.346,383.967,-136.796,173.187,45.853,159.095
C04352=1034.355,384.213,-136.838,173.195,45.857,159.097
C04353=1034.364,384.460,-136.880,173.202,45.861,159.099
C04354=1034.373,384.705,-136.922,173.211,45.864,159.100
C04355=1034.382,384.952,-136.964,173.219,45.868,159.102
C04356=1034.390,385.199,-137.006,173.228,45.871,159.104
C04357=1034.399,385.444,-137.049,173.236,45.875,159.106
C04358=1034.409,385.691,-137.091,173.245,45.878,159.108
C04359=1034.418,385.937,-137.133,173.252,45.882,159.110
C04360=1034.427,386.183,-137.175,173.260,45.885,159.111
C04361=1034.436,386.429,-137.217,173.269,45.889,159.113
C04362=1034.445,386.676,-137.259,173.277,45.892,159.115
C04363=1034.455,386.921,-137.301,173.286,45.896,159.117
C04364=1034.463,387.169,-137.344,173.295,45.899,159.119
C04365=1034.473,387.414,-137.387,173.303,45.903,159.121
C04366=1034.482,387.660,-137.429,173.311,45.906,159.123
C04367=1034.490,387.907,-137.471,173.320,45.910,159.125
C04368=1034.499,388.153,-137.514,173.328,45.914,159.126
C04369=1034.509,388.399,-137.557,173.336,45.918,159.128
C04370=1034.518,388.645,-137.600,173.345,45.922,159.130
C04371=1034.527,388.891,-137.642,173.353,45.925,159.132
C04372=1034.536,389.137,-137.684,173.362,45.929,159.134
C04373=1034.545,389.383,-137.728,173.370,45.932,159.136
C04374=1034.554,389.629,-137.770,173.379,45.937,159.138
C04375=1034.563,389.875,-137.813,173.388,45.940,159.140
C04376=1034.573,390.122,-137.856,173.396,45.944,159.142
C04377=1034.582,390.367,-137.899,173.405,45.948,159.144
C04378=1034.590,390.613,-137.942,173.414,45.952,159.146
C04379=1034.600,390.860,-137.984,173.422,45.955,159.148
C04380=1034.609,391.106,-138.027,173.431,45.959,159.150
C04381=1034.618,391.352,-138.071,173.441,45.963,159.152
C04382=1034.627,391.598,-138.114,173.449,45.967,159.154
C04383=1034.636,391.844,-138.157,173.458,45.971,159.156
C04384=1034.646,392.090,-138.200,173.467,45.975,159.158
C04385=1034.655,392.336,-138.243,173.475,45.979,159.160
C04386=1034.664,392.564,-138.283,173.484,45.982,159.162
C04387=1034.672,392.793,-138.324,173.492,45.986,159.164
C04388=1034.681,393.020,-138.364,173.500,45.990,159.165
C04389=1034.690,393.249,-138.404,173.509,45.993,159.167
C04390=1034.698,393.477,-138.445,173.516,45.997,159.169
C04391=1034.707,393.706,-138.485,173.525,46.001,159.171
C04392=1034.715,393.934,-138.525,173.533,46.004,159.173
C04393=1034.725,394.162,-138.565,173.542,46.008,159.175
C04394=1034.734,394.408,-138.608,173.551,46.012,159.177
C04395=1034.743,394.654,-138.652,173.560,46.017,159.179
C04396=1034.753,394.900,-138.696,173.568,46.020,159.181
C04397=1034.762,395.145,-138.740,173.578,46.024,159.183
C04398=1034.771,395.391,-138.784,173.587,46.029,159.185
C04399=1034.781,395.638,-138.828,173.596,46.033,159.188
C04400=1034.790,395.883,-138.870,173.605,46.037,159.190
C04401=1034.799,396.129,-138.914,173.615,46.041,159.192
C04402=1034.809,396.376,-138.959,173.624,46.046,159.194
C04403=1034.818,396.622,-139.003,173.633,46.050,159.196
C04404=1034.828,396.867,-139.046,173.643,46.054,159.198
C04405=1034.837,397.112,-139.091,173.652,46.058,159.200
C04406=1034.847,397.358,-139.135,173.661,46.062,159.203
C04407=1034.856,397.605,-139.179,173.670,46.066,159.205
C04408=1034.866,397.850,-139.222,173.680,46.071,159.207
C04409=1034.876,398.097,-139.267,173.690,46.075,159.209
C04410=1034.885,398.341,-139.311,173.699,46.079,159.211
C04411=1034.894,398.587,-139.355,173.707,46.084,159.213
C04412=1034.904,398.833,-139.399,173.718,46.088,159.216
C04413=1034.914,399.079,-139.443,173.727,46.092,159.218
C04414=1034.924,399.325,-139.488,173.736,46.096,159.220
C04415=1034.933,399.571,-139.532,173.746,46.101,159.222
C04416=1034.943,399.817,-139.576,173.756,46.105,159.225
C04417=1034.952,400.063,-139.621,173.765,46.110,159.227
C04418=1034.963,400.308,-139.665,173.775,46.115,159.229
C04419=1034.972,400.553,-139.710,173.784,46.119,159.232
C04420=1034.982,400.800,-139.754,173.794,46.123,159.234
C04421=1034.991,401.045,-139.799,173.803,46.128,159.236
C04422=1035.002,401.291,-139.844,173.813,46.132,159.238
C04423=1035.011,401.537,-139.889,173.824,46.137,159.241
C04424=1035.021,401.783,-139.933,173.833,46.141,159.243
C04425=1035.031,402.028,-139.977,173.843,46.146,159.245
C04426=1035.040,402.274,-140.022,173.852,46.151,159.248
C04427=1035.050,402.520,-140.067,173.863,46.155,159.250
C04428=1035.060,402.766,-140.112,173.873,46.160,159.253
C04429=1035.070,403.011,-140.157,173.882,46.164,159.255
C04430=1035.079,403.257,-140.203,173.892,46.169,159.257
C04431=1035.089,403.503,-140.247,173.903,46.173,159.260
C04432=1035.099,403.749,-140.293,173.912,46.178,159.262
C04433=1035.109,403.994,-140.337,173.922,46.183,159.264
C04434=1035.119,404.239,-140.383,173.933,46.188,159.267
C04435=1035.128,404.486,-140.429,173.942,46.193,159.269
C04436=1035.138,404.731,-140.474,173.952,46.197,159.272
C04437=1035.148,404.976,-140.519,173.963,46.202,159.274
C04438=1035.158,405.222,-140.564,173.973,46.207,159.277
C04439=1035.168,405.468,-140.609,173.983,46.211,159.279
C04440=1035.178,405.714,-140.656,173.993,46.216,159.282
C04441=1035.188,405.959,-140.700,174.003,46.221,159.284
C04442=1035.198,406.205,-140.746,174.013,46.226,159.287
C04443=1035.208,406.450,-140.791,174.024,46.231,159.289
C04444=1035.219,406.696,-140.837,174.034,46.236,159.291
C04445=1035.228,406.941,-140.883,174.045,46.241,159.294
C04446=1035.238,407.180,-140.927,174.054,46.245,159.296
C04447=1035.248,407.418,-140.971,174.065,46.250,159.299
C04448=1035.258,407.657,-141.016,174.075,46.255,159.301
C04449=1035.268,407.895,-141.060,174.085,46.260,159.304
C04450=1035.277,408.134,-141.105,174.095,46.265,159.306
C04451=1035.288,408.372,-141.150,174.105,46.270,159.309
C04452=1035.298,408.611,-141.194,174.116,46.274,159.311
C04453=1035.307,408.849,-141.238,174.126,46.279,159.314
C04454=1035.318,409.095,-141.284,174.137,46.284,159.316
C04455=1035.328,409.340,-141.330,174.147,46.289,159.319
C04456=1035.338,409.586,-141.376,174.158,46.294,159.322
C04457=1035.349,409.831,-141.422,174.168,46.299,159.324
C04458=1035.359,410.077,-141.468,174.179,46.305,159.327
C04459=1035.370,410.323,-141.514,174.190,46.310,159.330
C04460=1035.380,410.568,-141.561,174.201,46.314,159.332
C04461=1035.391,410.813,-141.607,174.212,46.320,159.335
C04462=1035.401,411.059,-141.653,174.223,46.325,159.338
C04463=1035.411,411.305,-141.699,174.233,46.330,159.340
C04464=1035.422,411.550,-141.746,174.244,46.335,159.343
C04465=1035.432,411.796,-141.793,174.255,46.341,159.346
C04466=1035.443,412.041,-141.839,174.267,46.346,159.348
C04467=1035.453,412.287,-141.886,174.278,46.351,159.351
C04468=1035.464,412.532,-141.932,174.289,46.357,159.354
C04469=1035.474,412.777,-141.980,174.299,46.362,159.357
C04470=1035.485,413.023,-142.025,174.311,46.367,159.359
C04471=1035.495,413.268,-142.073,174.322,46.373,159.362
C04472=1035.505,413.513,-142.120,174.333,46.378,159.365
C04473=1035.516,413.758,-142.166,174.345,46.383,159.368
C04474=1035.526,414.004,-142.213,174.356,46.389,159.371
C04475=1035.537,414.249,-142.260,174.366,46.394,159.373
C04476=1035.547,414.495,-142.307,174.378,46.400,159.376
C04477=1035.558,414.740,-142.354,174.389,46.405,159.379
C04478=1035.569,414.985,-142.401,174.401,46.410,159.382
C04479=1035.579,415.231,-142.448,174.412,46.416,159.385
C04480=1035.590,415.476,-142.495,174.424,46.422,159.388
C04481=1035.600,415.722,-142.542,174.435,46.427,159.391
C04482=1035.612,415.966,-142.590,174.447,46.433,159.394
C04483=1035.623,416.212,-142.637,174.458,46.438,159.396
C04484=1035.633,416.457,-142.684,174.470,46.444,159.399
C04485=1035.644,416.703,-142.732,174.481,46.450,159.402
C04486=1035.655,416.947,-142.779,174.493,46.455,159.405
C04487=1035.666,417.193,-142.826,174.506,46.461,159.408
C04488=1035.676,417.438,-142.874,174.517,46.467,159.411
C04489=1035.688,417.684,-142.922,174.529,46.472,159.414
C04490=1035.698,417.929,-142.969,174.541,46.477,159.417
C04491=1035.709,418.174,-143.018,174.552,46.484,159.420
C04492=1035.720,418.419,-143.065,174.564,46.489,159.423
C04493=1035.731,418.664,-143.113,174.577,46.495,159.426
C04494=1035.741,418.909,-143.160,174.588,46.501,159.429
C04495=1035.752,419.155,-143.209,174.600,46.507,159.432
C04496=1035.763,419.399,-143.257,174.612,46.512,159.435
C04497=1035.774,419.645,-143.305,174.625,46.518,159.438
C04498=1035.786,419.890,-143.353,174.637,46.524,159.442
C04499=1035.797,420.135,-143.401,174.649,46.530,159.445
C04500=1035.808,420.380,-143.449,174.661,46.536,159.448
C04501=1035.819,420.625,-143.497,174.673,46.542,159.451
C04502=1035.830,420.871,-143.545,174.685,46.548,159.454
C04503=1035.841,421.116,-143.594,174.698,46.554,159.457
C04504=1035.851,421.361,-143.642,174.710,46.560,159.460
C04505=1035.863,421.605,-143.690,174.723,46.566,159.463
C04506=1035.875,421.863,-143.741,174.735,46.573,159.467
C04507=1035.886,422.119,-143.792,174.749,46.579,159.470
C04508=1035.899,422.376,-143.842,174.762,46.585,159.473
C04509=1035.910,422.633,-143.893,174.775,46.591,159.477
C04510=1035.921,422.878,-143.942,174.788,46.597,159.480
C04511=1035.933,423.123,-143.990,174.801,46.604,159.483
C04512=1035.944,423.368,-144.038,174.813,46.610,159.487
C04513=1035.956,423.613,-144.087,174.826,46.616,159.490
C04514=1035.967,423.850,-144.135,174.838,46.622,159.493
C04515=1035.978,424.087,-144.183,174.851,46.628,159.496
C04516=1035.989,424.324,-144.230,174.863,46.634,159.499
C04517=1036.000,424.561,-144.277,174.876,46.640,159.503
C04518=1036.011,424.798,-144.325,174.888,46.647,159.506
C04519=1036.022,425.035,-144.373,174.901,46.653,159.509
C04520=1036.033,425.272,-144.420,174.913,46.658,159.512
C04521=1036.044,425.508,-144.467,174.926,46.665,159.516
C04522=1036.055,425.754,-144.517,174.940,46.671,159.519
C04523=1036.067,425.999,-144.566,174.953,46.678,159.523
C04524=1036.078,426.243,-144.615,174.965,46.684,159.526
C04525=1036.090,426.488,-144.665,174.979,46.690,159.529
C04526=1036.102,426.733,-144.714,174.992,46.697,159.533
C04527=1036.113,426.977,-144.764,175.006,46.703,159.536
C04528=1036.125,427.223,-144.813,175.019,46.710,159.540
C04529=1036.137,427.467,-144.862,175.033,46.716,159.543
C04530=1036.148,427.712,-144.913,175.046,46.723,159.547
C04531=1036.160,427.957,-144.962,175.060,46.730,159.550
C04532=1036.172,428.202,-145.012,175.073,46.736,159.554
C04533=1036.183,428.446,-145.062,175.087,46.743,159.557
C04534=1036.195,428.691,-145.112,175.101,46.749,159.561
C04535=1036.207,428.936,-145.161,175.114,46.756,159.565
C04536=1036.218,429.181,-145.212,175.128,46.763,159.568
C04537=1036.230,429.425,-145.262,175.142,46.770,159.572
C04538=1036.242,429.670,-145.312,175.156,46.776,159.575
C04539=1036.253,429.915,-145.362,175.169,46.783,159.579
C04540=1036.266,430.159,-145.412,175.183,46.790,159.583
C04541=1036.278,430.404,-145.462,175.197,46.796,159.586
C04542=1036.290,430.649,-145.514,175.212,46.803,159.590
C04543=1036.302,430.893,-145.563,175.226,46.810,159.594
C04544=1036.314,431.138,-145.613,175.240,46.817,159.598
C04545=1036.326,431.383,-145.664,175.254,46.824,159.601
C04546=1036.338,431.627,-145.715,175.268,46.831,159.605
C04547=1036.350,431.872,-145.765,175.282,46.838,159.609
C04548=1036.362,432.116,-145.816,175.296,46.845,159.613
C04549=1036.374,432.360,-145.866,175.311,46.852,159.616
C04550=1036.387,432.605,-145.917,175.326,46.859,159.620
C04551=1036.398,432.850,-145.968,175.341,46.865,159.624
C04552=1036.411,433.094,-146.019,175.355,46.872,159.628
C04553=1036.423,433.338,-146.069,175.369,46.880,159.632
C04554=1036.435,433.583,-146.121,175.384,46.887,159.635
C04555=1036.449,433.828,-146.172,175.398,46.894,159.639
C04556=1036.461,434.072,-146.222,175.414,46.901,159.643
C04557=1036.473,434.317,-146.273,175.428,46.908,159.647
C04558=1036.485,434.561,-146.324,175.443,46.915,159.651
C04559=1036.497,434.806,-146.376,175.458,46.922,159.655
C04560=1036.511,435.050,-146.428,175.473,46.929,159.659
C04561=1036.523,435.294,-146.479,175.488,46.937,159.663
C04562=1036.535,435.539,-146.530,175.503,46.944,159.667
C04563=1036.547,435.782,-146.582,175.518,46.952,159.671
C04564=1036.560,436.028,-146.634,175.533,46.959,159.675
C04565=1036.573,436.272,-146.684,175.549,46.966,159.679
C04566=1036.585,436.516,-146.737,175.564,46.974,159.683
C04567=1036.598,436.759,-146.788,175.579,46.981,159.687
C04568=1036.611,437.003,-146.840,175.595,46.988,159.692
C04569=1036.623,437.247,-146.892,175.610,46.996,159.696
C04570=1036.636,437.490,-146.943,175.626,47.003,159.700
C04571=1036.648,437.734,-146.995,175.641,47.011,159.704
C04572=1036.661,437.979,-147.047,175.657,47.018,159.708
C04573=1036.674,438.222,-147.099,175.673,47.025,159.712
C04574=1036.687,438.466,-147.151,175.689,47.033,159.717
C04575=1036.699,438.711,-147.203,175.704,47.041,159.721
C04576=1036.712,438.955,-147.256,175.720,47.049,159.725
C04577=1036.725,439.199,-147.307,175.736,47.056,159.729
C04578=1036.738,439.443,-147.360,175.752,47.064,159.734
C04579=1036.751,439.687,-147.413,175.768,47.072,159.738
C04580=1036.764,439.932,-147.465,175.784,47.079,159.742
C04581=1036.777,440.175,-147.517,175.801,47.087,159.747
C04582=1036.790,440.419,-147.570,175.817,47.094,159.751
C04583=1036.803,440.664,-147.623,175.833,47.102,159.755
C04584=1036.816,440.908,-147.676,175.849,47.110,159.760
C04585=1036.829,441.152,-147.729,175.866,47.118,159.764
C04586=1036.842,441.396,-147.781,175.882,47.126,159.769
C04587=1036.855,441.640,-147.834,175.898,47.134,159.773
C04588=1036.868,441.884,-147.888,175.916,47.142,159.778
C04589=1036.882,442.128,-147.941,175.932,47.150,159.782
C04590=1036.895,442.372,-147.993,175.948,47.158,159.787
C04591=1036.908,442.616,-148.047,175.965,47.166,159.791
C04592=1036.922,442.860,-148.100,175.982,47.174,159.796
C04593=1036.935,443.104,-148.153,175.999,47.182,159.800
C04594=1036.949,443.347,-148.206,176.017,47.190,159.805
C04595=1036.963,443.591,-148.260,176.033,47.198,159.810
C04596=1036.976,443.835,-148.313,176.051,47.206,159.814
C04597=1036.989,444.079,-148.367,176.067,47.214,159.819
C04598=1037.003,444.322,-148.420,176.085,47.222,159.824
C04599=1037.017,444.564,-148.472,176.101,47.230,159.828
C04600=1037.032,444.808,-148.524,176.119,47.238,159.833
C04601=1037.047,445.053,-148.577,176.137,47.246,159.837
C04602=1037.064,445.295,-148.628,176.154,47.254,159.842
C04603=1037.080,445.539,-148.679,176.172,47.261,159.846
C04604=1037.097,445.783,-148.729,176.190,47.269,159.851
C04605=1037.114,446.027,-148.779,176.208,47.276,159.856
C04606=1037.132,446.271,-148.829,176.225,47.284,159.860
C04607=1037.151,446.514,-148.878,176.243,47.291,159.865
C04608=1037.170,446.758,-148.927,176.262,47.298,159.869
C04609=1037.190,447.003,-148.976,176.279,47.305,159.874
C04610=1037.210,447.247,-149.023,176.297,47.312,159.878
C04611=1037.231,447.492,-149.070,176.316,47.319,159.883
C04612=1037.253,447.736,-149.117,176.334,47.325,159.887
C04613=1037.275,447.981,-149.164,176.353,47.332,159.892
C04614=1037.297,448.225,-149.210,176.371,47.339,159.896
C04615=1037.320,448.470,-149.256,176.390,47.346,159.901
C04616=1037.344,448.715,-149.301,176.409,47.352,159.905
C04617=1037.368,448.960,-149.346,176.428,47.358,159.909
C04618=1037.392,449.205,-149.390,176.446,47.365,159.914
C04619=1037.418,449.450,-149.434,176.465,47.371,159.918
C04620=1037.443,449.695,-149.477,176.484,47.377,159.923
C04621=1037.470,449.939,-149.520,176.503,47.383,159.927
C04622=1037.497,450.185,-149.563,176.523,47.389,159.931
C04623=1037.524,450.430,-149.604,176.542,47.395,159.936
C04624=1037.552,450.676,-149.647,176.561,47.401,159.940
C04625=1037.580,450.921,-149.687,176.580,47.406,159.944
C04626=1037.620,451.251,-149.742,176.606,47.414,159.950
C04627=1037.660,451.580,-149.795,176.633,47.421,159.956
C04628=1037.700,451.908,-149.848,176.660,47.428,159.962
C04629=1037.742,452.237,-149.900,176.686,47.436,159.967
C04630=1037.451,452.292,-150.223,176.689,47.507,159.990
C04631=1037.411,451.977,-150.174,176.663,47.501,159.984
C04632=1037.372,451.661,-150.123,176.638,47.494,159.979
C04633=1037.332,451.346,-150.072,176.613,47.487,159.973
C04634=1037.295,451.030,-150.020,176.588,47.479,159.968
C04635=1037.266,450.785,-149.979,176.568,47.474,159.963
C04636=1037.237,450.539,-149.938,176.548,47.469,159.959
C04637=1037.210,450.294,-149.896,176.529,47.462,159.955
C04638=1037.183,450.048,-149.853,176.510,47.457,159.950
C04639=1037.156,449.803,-149.811,176.490,47.451,159.946
C04640=1037.130,449.558,-149.768,176.471,47.445,159.942
C04641=1037.105,449.314,-149.725,176.452,47.439,159.937
C04642=1037.079,449.069,-149.680,176.433,47.433,159.933
C04643=1037.055,448.823,-149.636,176.415,47.426,159.928
C04644=1037.031,448.579,-149.591,176.396,47.420,159.924
C04645=1037.008,448.334,-149.546,176.377,47.414,159.920
C04646=1036.985,448.089,-149.499,176.359,47.407,159.915
C04647=1036.963,447.845,-149.454,176.340,47.401,159.911
C04648=1036.941,447.601,-149.407,176.321,47.394,159.906
C04649=1036.920,447.355,-149.360,176.303,47.387,159.902
C04650=1036.899,447.111,-149.312,176.285,47.380,159.897
C04651=1036.879,446.867,-149.263,176.267,47.374,159.893
C04652=1036.860,446.622,-149.215,176.248,47.367,159.888
C04653=1036.841,446.378,-149.166,176.231,47.359,159.884
C04654=1036.822,446.135,-149.117,176.212,47.352,159.879
C04655=1036.805,445.891,-149.067,176.195,47.345,159.875
C04656=1036.787,445.646,-149.017,176.176,47.338,159.870
C04657=1036.770,445.403,-148.966,176.159,47.330,159.865
C04658=1036.754,445.160,-148.915,176.142,47.323,159.861
C04659=1036.739,444.916,-148.864,176.124,47.315,159.856
C04660=1036.723,444.672,-148.811,176.106,47.307,159.852
C04661=1036.709,444.429,-148.759,176.089,47.300,159.847
C04662=1036.694,444.187,-148.706,176.072,47.291,159.842
C04663=1036.681,443.943,-148.653,176.055,47.283,159.838
C04664=1036.666,443.699,-148.599,176.037,47.276,159.833
C04665=1036.653,443.456,-148.546,176.020,47.267,159.828
C04666=1036.640,443.212,-148.493,176.003,47.260,159.824
C04667=1036.627,442.968,-148.439,175.986,47.251,159.819
C04668=1036.613,442.725,-148.386,175.970,47.243,159.815
C04669=1036.600,442.481,-148.333,175.952,47.236,159.810
C04670=1036.586,442.236,-148.280,175.936,47.227,159.806
C04671=1036.573,441.992,-148.227,175.918,47.220,159.801
C04672=1036.559,441.748,-148.174,175.902,47.212,159.797
C04673=1036.546,441.504,-148.121,175.886,47.204,159.792
C04674=1036.533,441.260,-148.068,175.869,47.196,159.788
C04675=1036.521,441.016,-148.015,175.852,47.189,159.783
C04676=1036.508,440.772,-147.962,175.836,47.181,159.779
C04677=1036.494,440.528,-147.910,175.819,47.173,159.774
C04678=1036.481,440.284,-147.857,175.803,47.166,159.770
C04679=1036.468,440.040,-147.805,175.787,47.158,159.766
C04680=1036.455,439.796,-147.751,175.771,47.150,159.761
C04681=1036.442,439.551,-147.699,175.754,47.142,159.757
C04682=1036.430,439.307,-147.647,175.738,47.135,159.753
C04683=1036.416,439.064,-147.594,175.722,47.127,159.748
C04684=1036.403,438.819,-147.542,175.706,47.120,159.744
C04685=1036.391,438.575,-147.490,175.690,47.112,159.740
C04686=1036.378,438.331,-147.438,175.675,47.105,159.736
C04687=1036.364,438.086,-147.386,175.659,47.097,159.732
C04688=1036.352,437.843,-147.334,175.643,47.090,159.727
C04689=1036.339,437.598,-147.281,175.628,47.083,159.723
C04690=1036.327,437.354,-147.230,175.613,47.075,159.719
C04691=1036.314,437.109,-147.178,175.597,47.067,159.715
C04692=1036.301,436.865,-147.125,175.581,47.060,159.711
C04693=1036.289,436.619,-147.074,175.566,47.053,159.707
C04694=1036.276,436.374,-147.022,175.550,47.046,159.703
C04695=1036.263,436.131,-146.970,175.535,47.039,159.698
C04696=1036.251,435.886,-146.919,175.519,47.031,159.694
C04697=1036.238,435.642,-146.867,175.504,47.024,159.690
C04698=1036.226,435.397,-146.816,175.489,47.017,159.686
C04699=1036.213,435.153,-146.765,175.474,47.009,159.682
C04700=1036.201,434.909,-146.713,175.459,47.002,159.678
C04701=1036.189,434.665,-146.662,175.444,46.995,159.674
C04702=1036.176,434.420,-146.610,175.429,46.988,159.670
C04703=1036.164,434.176,-146.559,175.414,46.981,159.667
C04704=1036.151,433.931,-146.508,175.399,46.974,159.663
C04705=1036.139,433.687,-146.457,175.385,46.967,159.659
C04706=1036.127,433.442,-146.407,175.370,46.960,159.655
C04707=1036.114,433.198,-146.356,175.355,46.953,159.651
C04708=1036.102,432.953,-146.305,175.341,46.946,159.647
C04709=1036.090,432.709,-146.254,175.326,46.939,159.643
C04710=1036.077,432.464,-146.204,175.312,46.932,159.639
C04711=1036.065,432.220,-146.152,175.297,46.926,159.636
C04712=1036.053,431.975,-146.102,175.282,46.919,159.632
C04713=1036.040,431.731,-146.052,175.268,46.912,159.628
C04714=1036.029,431.486,-146.001,175.254,46.905,159.624
C04715=1036.017,431.241,-145.951,175.239,46.898,159.621
C04716=1036.004,430.997,-145.900,175.225,46.891,159.617
C04717=1035.993,430.752,-145.850,175.211,46.884,159.613
C04718=1035.981,430.507,-145.800,175.197,46.877,159.609
C04719=1035.968,430.263,-145.749,175.183,46.871,159.606
C04720=1035.957,430.018,-145.698,175.169,46.864,159.602
C04721=1035.945,429.774,-145.648,175.155,46.857,159.598
C04722=1035.932,429.529,-145.598,175.141,46.851,159.595
C04723=1035.921,429.284,-145.548,175.127,46.844,159.591
C04724=1035.909,429.040,-145.498,175.114,46.837,159.588
C04725=1035.897,428.794,-145.448,175.100,46.831,159.584
C04726=1035.886,428.550,-145.398,175.086,46.825,159.580
C04727=1035.874,428.305,-145.348,175.072,46.817,159.577
C04728=1035.862,428.061,-145.298,175.058,46.811,159.573
C04729=1035.851,427.815,-145.248,175.044,46.805,159.570
C04730=1035.839,427.571,-145.199,175.032,46.798,159.566
C04731=1035.827,427.326,-145.149,175.018,46.792,159.563
C04732=1035.815,427.082,-145.099,175.005,46.785,159.559
C04733=1035.803,426.836,-145.050,174.991,46.779,159.556
C04734=1035.793,426.591,-145.000,174.978,46.772,159.552
C04735=1035.781,426.346,-144.950,174.964,46.766,159.549
C04736=1035.769,426.102,-144.901,174.951,46.760,159.545
C04737=1035.758,425.857,-144.852,174.937,46.753,159.542
C04738=1035.746,425.612,-144.803,174.925,46.747,159.539
C04739=1035.734,425.367,-144.754,174.911,46.741,159.535
C04740=1035.723,425.122,-144.705,174.898,46.735,159.532
C04741=1035.711,424.877,-144.656,174.886,46.728,159.529
C04742=1035.700,424.632,-144.607,174.872,46.722,159.525
C04743=1035.689,424.388,-144.558,174.859,46.716,159.522
C04744=1035.677,424.143,-144.509,174.847,46.710,159.518
C04745=1035.665,423.897,-144.459,174.834,46.703,159.515
C04746=1035.655,423.652,-144.410,174.820,46.697,159.512
C04747=1035.643,423.409,-144.362,174.808,46.691,159.509
C04748=1035.632,423.165,-144.313,174.795,46.685,159.505
C04749=1035.621,422.921,-144.265,174.782,46.679,159.502
C04750=1035.609,422.677,-144.217,174.770,46.673,159.499
C04751=1035.598,422.432,-144.168,174.758,46.667,159.496
C04752=1035.586,422.189,-144.120,174.745,46.661,159.492
C04753=1035.575,421.945,-144.071,174.732,46.655,159.489
C04754=1035.564,421.700,-144.024,174.719,46.649,159.486
C04755=1035.553,421.456,-143.975,174.707,46.644,159.483
C04756=1035.542,421.210,-143.927,174.694,46.637,159.480
C04757=1035.531,420.965,-143.878,174.682,46.632,159.477
C04758=1035.520,420.720,-143.830,174.670,46.626,159.473
C04759=1035.509,420.475,-143.782,174.657,46.620,159.470
C04760=1035.497,420.230,-143.734,174.646,46.614,159.467
C04761=1035.486,419.984,-143.686,174.634,46.608,159.464
C04762=1035.476,419.740,-143.638,174.621,46.602,159.461
C04763=1035.464,419.494,-143.590,174.609,46.597,159.458
C04764=1035.453,419.249,-143.542,174.597,46.591,159.455
C04765=1035.443,419.004,-143.494,174.584,46.585,159.452
C04766=1035.432,418.759,-143.445,174.572,46.579,159.449
C04767=1035.420,418.514,-143.398,174.561,46.573,159.446
C04768=1035.410,418.269,-143.351,174.549,46.568,159.443
C04769=1035.399,418.023,-143.302,174.536,46.562,159.440
C04770=1035.388,417.779,-143.254,174.524,46.556,159.437
C04771=1035.377,417.533,-143.207,174.513,46.551,159.434
C04772=1035.367,417.288,-143.159,174.501,46.545,159.431
C04773=1035.355,417.042,-143.112,174.489,46.539,159.428
C04774=1035.345,416.797,-143.065,174.478,46.534,159.425
C04775=1035.329,416.454,-142.998,174.461,46.526,159.421
C04776=1035.314,416.111,-142.931,174.444,46.518,159.417
C04777=1035.300,415.767,-142.866,174.429,46.511,159.413
C04778=1035.284,415.424,-142.800,174.412,46.503,159.408
C04779=1035.274,415.179,-142.752,174.401,46.498,159.406
C04780=1035.262,414.933,-142.705,174.389,46.492,159.403
C04781=1035.252,414.688,-142.658,174.378,46.487,159.400
C04782=1035.241,414.443,-142.611,174.366,46.482,159.397
C04783=1035.231,414.198,-142.564,174.355,46.476,159.394
C04784=1035.220,413.951,-142.517,174.343,46.471,159.391
C04785=1035.210,413.706,-142.471,174.333,46.465,159.389
C04786=1035.199,413.461,-142.423,174.322,46.460,159.386
C04787=1035.188,413.216,-142.377,174.310,46.455,159.383
C04788=1035.178,412.971,-142.330,174.299,46.449,159.380
C04789=1035.168,412.725,-142.284,174.288,46.444,159.378
C04790=1035.157,412.480,-142.237,174.276,46.439,159.375
C04791=1035.147,412.234,-142.191,174.265,46.433,159.372
C04792=1035.137,411.989,-142.143,174.255,46.428,159.369
C04793=1035.126,411.744,-142.097,174.243,46.423,159.367
C04794=1035.116,411.498,-142.050,174.232,46.418,159.364
C04795=1035.106,411.252,-142.004,174.221,46.413,159.361
C04796=1035.095,411.007,-141.957,174.211,46.408,159.358
C04797=1035.084,410.761,-141.911,174.199,46.403,159.356
C04798=1035.074,410.516,-141.865,174.188,46.397,159.353
C04799=1035.064,410.270,-141.819,174.178,46.392,159.350
C04800=1035.053,410.025,-141.772,174.167,46.387,159.348
C04801=1035.042,409.779,-141.726,174.156,46.382,159.345
C04802=1035.032,409.534,-141.680,174.146,46.377,159.343
C04803=1035.022,409.288,-141.634,174.135,46.372,159.340
C04804=1035.012,409.043,-141.588,174.124,46.368,159.337
C04805=1035.001,408.797,-141.542,174.113,46.363,159.335
C04806=1034.990,408.552,-141.497,174.102,46.358,159.332
C04807=1034.975,408.170,-141.426,174.086,46.350,159.328
C04808=1034.959,407.790,-141.355,174.069,46.342,159.324
C04809=1034.943,407.409,-141.283,174.054,46.335,159.320
C04810=1034.928,407.028,-141.213,174.038,46.327,159.316
C04811=1034.918,406.782,-141.167,174.027,46.322,159.314
C04812=1034.907,406.536,-141.122,174.017,46.318,159.311
C04813=1034.897,406.291,-141.076,174.006,46.313,159.309
C04814=1034.887,406.045,-141.031,173.996,46.308,159.306
C04815=1034.878,405.800,-140.985,173.985,46.303,159.304
C04816=1034.867,405.554,-140.940,173.975,46.299,159.301
C04817=1034.857,405.309,-140.894,173.966,46.294,159.299
C04818=1034.848,405.063,-140.849,173.955,46.289,159.296
C04819=1034.837,404.818,-140.803,173.945,46.285,159.294
C04820=1034.827,404.572,-140.758,173.935,46.280,159.292
C04821=1034.818,404.326,-140.713,173.924,46.275,159.289
C04822=1034.808,404.080,-140.668,173.915,46.270,159.287
C04823=1034.798,403.835,-140.622,173.905,46.266,159.284
C04824=1034.788,403.589,-140.577,173.894,46.261,159.282
C04825=1034.778,403.343,-140.532,173.884,46.257,159.280
C04826=1034.769,403.098,-140.487,173.875,46.252,159.277
C04827=1034.759,402.852,-140.442,173.865,46.247,159.275
C04828=1034.749,402.606,-140.397,173.854,46.243,159.272
C04829=1034.739,402.360,-140.352,173.845,46.238,159.270
C04830=1034.729,402.115,-140.307,173.835,46.234,159.268
C04831=1034.720,401.869,-140.262,173.825,46.229,159.265
C04832=1034.710,401.624,-140.218,173.816,46.225,159.263
C04833=1034.700,401.377,-140.173,173.805,46.220,159.261
C04834=1034.690,401.131,-140.128,173.795,46.216,159.258
C04835=1034.681,400.886,-140.083,173.786,46.211,159.256
C04836=1034.671,400.640,-140.039,173.776,46.207,159.254
C04837=1034.662,400.394,-139.995,173.767,46.202,159.252
C04838=1034.652,400.149,-139.950,173.757,46.198,159.249
C04839=1034.642,399.903,-139.906,173.747,46.194,159.247
C04840=1034.632,399.657,-139.861,173.738,46.190,159.245
C04841=1034.623,399.411,-139.817,173.728,46.185,159.242
C04842=1034.613,399.166,-139.772,173.718,46.181,159.240
C04843=1034.603,398.920,-139.728,173.709,46.177,159.238
C04844=1034.594,398.674,-139.683,173.699,46.172,159.236
C04845=1034.584,398.428,-139.640,173.690,46.168,159.234
C04846=1034.574,398.182,-139.596,173.680,46.164,159.231
C04847=1034.564,397.937,-139.551,173.671,46.160,159.229
C04848=1034.555,397.691,-139.507,173.661,46.156,159.227
C04849=1034.545,397.445,-139.464,173.652,46.151,159.225
C04850=1034.536,397.199,-139.420,173.643,46.148,159.223
C04851=1034.527,396.953,-139.376,173.634,46.143,159.221
C04852=1034.517,396.707,-139.331,173.625,46.139,159.218
C04853=1034.507,396.461,-139.288,173.615,46.135,159.216
C04854=1034.498,396.216,-139.244,173.606,46.131,159.214
C04855=1034.489,395.970,-139.200,173.597,46.127,159.212
C04856=1034.479,395.724,-139.157,173.587,46.123,159.210
C04857=1034.469,395.478,-139.112,173.578,46.118,159.208
C04858=1034.460,395.232,-139.069,173.569,46.114,159.205
C04859=1034.451,394.986,-139.025,173.559,46.110,159.203
C04860=1034.441,394.740,-138.981,173.550,46.106,159.201
C04861=1034.432,394.495,-138.937,173.542,46.102,159.199
C04862=1034.423,394.248,-138.894,173.533,46.098,159.197
C04863=1034.414,394.019,-138.853,173.524,46.094,159.195
C04864=1034.405,393.790,-138.813,173.516,46.091,159.193
C04865=1034.397,393.560,-138.773,173.507,46.087,159.191
C04866=1034.388,393.331,-138.732,173.498,46.084,159.189
C04867=1034.379,393.101,-138.691,173.490,46.080,159.188
C04868=1034.370,392.872,-138.651,173.482,46.076,159.186
C04869=1034.362,392.643,-138.611,173.474,46.072,159.184
C04870=1034.353,392.414,-138.570,173.465,46.069,159.182
C04871=1034.343,392.167,-138.528,173.456,46.065,159.180
C04872=1034.335,391.922,-138.484,173.448,46.061,159.178
C04873=1034.325,391.676,-138.441,173.439,46.057,159.176
C04874=1034.316,391.430,-138.398,173.430,46.053,159.174
C04875=1034.306,391.183,-138.355,173.420,46.050,159.172
C04876=1034.298,390.938,-138.311,173.412,46.046,159.170
C04877=1034.289,390.692,-138.268,173.403,46.042,159.168
C04878=1034.279,390.445,-138.226,173.395,46.038,159.166
C04879=1034.270,390.199,-138.183,173.386,46.035,159.164
C04880=1034.261,389.953,-138.140,173.377,46.031,159.162
C04881=1034.252,389.707,-138.097,173.369,46.027,159.160
C04882=1034.243,389.461,-138.054,173.360,46.024,159.158
C04883=1034.234,389.215,-138.012,173.352,46.020,159.156
C04884=1034.224,388.969,-137.969,173.343,46.016,159.154
C04885=1034.216,388.723,-137.926,173.334,46.012,159.152
C04886=1034.206,388.477,-137.884,173.326,46.009,159.150
C04887=1034.197,388.230,-137.840,173.317,46.005,159.148
C04888=1034.188,387.984,-137.798,173.309,46.002,159.147
C04889=1034.179,387.739,-137.755,173.300,45.998,159.145
C04890=1034.171,387.492,-137.713,173.292,45.994,159.143
C04891=1034.161,387.246,-137.671,173.283,45.990,159.141
C04892=1034.151,387.000,-137.628,173.275,45.987,159.139
C04893=1034.143,386.753,-137.586,173.266,45.984,159.137
C04894=1034.133,386.508,-137.544,173.258,45.980,159.135
C04895=1034.124,386.261,-137.502,173.249,45.977,159.134
C04896=1034.116,386.015,-137.459,173.242,45.973,159.132
C04897=1034.106,385.768,-137.417,173.233,45.969,159.130
C04898=1034.097,385.522,-137.374,173.225,45.966,159.128
C04899=1034.088,385.276,-137.333,173.216,45.963,159.126
C04900=1034.079,385.030,-137.291,173.208,45.959,159.124
C04901=1034.070,384.784,-137.249,173.200,45.956,159.123
C04902=1034.061,384.538,-137.207,173.191,45.952,159.121
C04903=1034.052,384.291,-137.165,173.184,45.949,159.119
C04904=1034.043,384.045,-137.123,173.175,45.946,159.117
C04905=1034.035,383.799,-137.080,173.167,45.943,159.116
C04906=1034.026,383.552,-137.039,173.158,45.939,159.114
C04907=1034.017,383.306,-136.997,173.150,45.936,159.112
C04908=1034.008,383.060,-136.955,173.143,45.932,159.110
C04909=1033.999,382.813,-136.914,173.135,45.929,159.108
C04910=1033.990,382.567,-136.872,173.126,45.926,159.107
C04911=1033.981,382.321,-136.829,173.118,45.923,159.105
C04912=1033.972,382.076,-136.788,173.111,45.919,159.103
C04913=1033.963,381.829,-136.746,173.102,45.916,159.102
C04914=1033.955,381.582,-136.705,173.094,45.913,159.100
C04915=1033.946,381.336,-136.664,173.087,45.909,159.098
C04916=1033.938,381.089,-136.621,173.078,45.906,159.096
C04917=1033.929,380.843,-136.580,173.070,45.903,159.095
C04918=1033.920,380.597,-136.538,173.062,45.900,159.093
C04919=1033.912,380.351,-136.497,173.054,45.896,159.091
C04920=1033.903,380.104,-136.455,173.046,45.894,159.090
C04921=1033.894,379.857,-136.414,173.039,45.890,159.088
C04922=1033.886,379.612,-136.372,173.031,45.887,159.086
C04923=1033.878,379.399,-136.336,173.024,45.884,159.085
C04924=1033.870,379.188,-136.301,173.017,45.882,159.083
C04925=1033.863,378.976,-136.265,173.011,45.879,159.082
C04926=1033.857,378.764,-136.230,173.004,45.876,159.080
C04927=1033.848,378.552,-136.194,172.997,45.873,159.079
C04928=1033.841,378.340,-136.158,172.990,45.871,159.077
C04929=1033.834,378.129,-136.123,172.984,45.868,159.076
C04930=1033.827,377.917,-136.088,172.978,45.865,159.075
C04931=1033.818,377.670,-136.046,172.970,45.862,159.073
C04932=1033.809,377.424,-136.006,172.961,45.859,159.071
C04933=1033.801,377.177,-135.965,172.954,45.856,159.070
C04934=1033.792,376.931,-135.923,172.946,45.853,159.068
C04935=1033.783,376.684,-135.882,172.939,45.850,159.067
C04936=1033.774,376.438,-135.842,172.931,45.848,159.065
C04937=1033.766,376.191,-135.801,172.924,45.844,159.063
C04938=1033.757,375.945,-135.760,172.916,45.841,159.062
C04939=1033.749,375.698,-135.719,172.909,45.839,159.060
C04940=1033.740,375.452,-135.679,172.901,45.836,159.059
C04941=1033.731,375.205,-135.638,172.893,45.832,159.057
C04942=1033.723,374.959,-135.597,172.885,45.830,159.056
C04943=1033.715,374.712,-135.556,172.878,45.827,159.054
C04944=1033.706,374.466,-135.516,172.870,45.824,159.052
C04945=1033.697,374.219,-135.475,172.863,45.821,159.051
C04946=1033.689,373.973,-135.435,172.856,45.818,159.049
C04947=1033.680,373.726,-135.394,172.848,45.816,159.048
C04948=1033.672,373.480,-135.354,172.841,45.812,159.046
C04949=1033.664,373.234,-135.313,172.833,45.810,159.045
C04950=1033.655,372.987,-135.272,172.826,45.807,159.043
C04951=1033.646,372.741,-135.232,172.819,45.804,159.042
C04952=1033.638,372.495,-135.191,172.811,45.801,159.040
C04953=1033.630,372.247,-135.151,172.804,45.799,159.039
C04954=1033.621,372.001,-135.111,172.796,45.796,159.037
C04955=1033.613,371.755,-135.070,172.789,45.793,159.036
C04956=1033.605,371.508,-135.029,172.782,45.790,159.034
C04957=1033.597,371.261,-134.990,172.774,45.788,159.033
C04958=1033.588,371.015,-134.949,172.767,45.785,159.031
C04959=1033.580,370.768,-134.909,172.760,45.782,159.030
C04960=1033.572,370.521,-134.869,172.754,45.779,159.028
C04961=1033.563,370.275,-134.829,172.746,45.777,159.027
C04962=1033.555,370.028,-134.789,172.739,45.774,159.025
C04963=1033.547,369.782,-134.748,172.732,45.771,159.024
C04964=1033.539,369.535,-134.709,172.724,45.769,159.022
C04965=1033.530,369.288,-134.668,172.717,45.766,159.021
C04966=1033.522,369.042,-134.628,172.710,45.764,159.020
C04967=1033.514,368.795,-134.588,172.703,45.761,159.018
C04968=1033.505,368.549,-134.548,172.696,45.758,159.017
C04969=1033.497,368.302,-134.509,172.689,45.756,159.015
C04970=1033.489,368.055,-134.469,172.682,45.753,159.014
C04971=1033.480,367.808,-134.429,172.675,45.750,159.012
C04972=1033.471,367.562,-134.389,172.667,45.748,159.011
C04973=1033.463,367.315,-134.349,172.660,45.745,159.010
C04974=1033.455,367.068,-134.310,172.654,45.743,159.008
C04975=1033.447,366.821,-134.270,172.647,45.741,159.007
C04976=1033.439,366.575,-134.231,172.640,45.738,159.005
C04977=1033.430,366.328,-134.192,172.632,45.735,159.004
C04978=1033.423,366.081,-134.152,172.625,45.733,159.003
C04979=1033.414,365.835,-134.112,172.619,45.731,159.001
C04980=1033.406,365.588,-134.073,172.612,45.728,159.000
C04981=1033.398,365.341,-134.033,172.605,45.725,158.999
C04982=1033.390,365.095,-133.994,172.598,45.723,158.997
C04983=1033.376,364.692,-133.928,172.586,45.719,158.995
C04984=1033.363,364.289,-133.864,172.576,45.715,158.993
C04985=1033.350,363.886,-133.801,172.565,45.711,158.991
C04986=1033.336,363.482,-133.736,172.553,45.708,158.988
C04987=1033.328,363.236,-133.697,172.546,45.705,158.987
C04988=1033.321,362.990,-133.657,172.540,45.703,158.986
C04989=1033.313,362.742,-133.619,172.533,45.700,158.985
C04990=1033.305,362.495,-133.579,172.526,45.698,158.983
C04991=1033.296,362.249,-133.539,172.519,45.696,158.982
C04992=1033.288,362.002,-133.501,172.513,45.693,158.981
C04993=1033.281,361.755,-133.461,172.506,45.691,158.979
C04994=1033.273,361.509,-133.422,172.499,45.689,158.978
C04995=1033.265,361.262,-133.383,172.493,45.686,158.977
C04996=1033.256,361.015,-133.344,172.486,45.684,158.975
C04997=1033.249,360.768,-133.306,172.480,45.682,158.974
C04998=1033.240,360.521,-133.267,172.473,45.680,158.973
C04999=1033.233,360.274,-133.227,172.466,45.677,158.972
C05000=1033.225,360.027,-133.189,172.459,45.675,158.970
C05001=1033.217,359.781,-133.150,172.453,45.673,158.969
C05002=1033.209,359.534,-133.111,172.446,45.671,158.968
C05003=1033.200,359.287,-133.072,172.440,45.668,158.967
C05004=1033.192,359.040,-133.034,172.433,45.667,158.965
C05005=1033.184,358.794,-132.995,172.427,45.664,158.964
C05006=1033.176,358.547,-132.956,172.420,45.663,158.963
C05007=1033.168,358.299,-132.918,172.413,45.660,158.962
C05008=1033.160,358.053,-132.879,172.407,45.658,158.961
C05009=1033.152,357.806,-132.841,172.400,45.656,158.959
C05010=1033.144,357.558,-132.802,172.394,45.654,158.958
C05011=1033.137,357.312,-132.764,172.387,45.652,158.957
C05012=1033.128,357.065,-132.725,172.381,45.650,158.956
C05013=1033.121,356.819,-132.686,172.374,45.648,158.954
C05014=1033.112,356.572,-132.648,172.368,45.646,158.953
C05015=1033.105,356.325,-132.609,172.362,45.643,158.952
C05016=1033.097,356.078,-132.571,172.356,45.641,158.951
C05017=1033.089,355.831,-132.532,172.349,45.640,158.950
C05018=1033.081,355.583,-132.495,172.342,45.637,158.948
C05019=1033.073,355.336,-132.456,172.336,45.635,158.947
C05020=1033.066,355.090,-132.418,172.330,45.634,158.946
C05021=1033.058,354.842,-132.379,172.323,45.631,158.945
C05022=1033.049,354.596,-132.342,172.317,45.629,158.944
C05023=1033.041,354.348,-132.304,172.311,45.627,158.943
C05024=1033.034,354.102,-132.265,172.305,45.626,158.941
C05025=1033.026,353.855,-132.227,172.298,45.624,158.940
C05026=1033.018,353.608,-132.189,172.292,45.622,158.939
C05027=1033.011,353.361,-132.151,172.285,45.620,158.938
C05028=1033.002,353.114,-132.113,172.279,45.618,158.937
C05029=1032.995,352.867,-132.076,172.273,45.616,158.936
C05030=1032.987,352.620,-132.037,172.267,45.614,158.935
C05031=1032.979,352.373,-131.999,172.261,45.612,158.933
C05032=1032.972,352.126,-131.961,172.254,45.610,158.932
C05033=1032.963,351.879,-131.923,172.248,45.609,158.931
C05034=1032.956,351.632,-131.886,172.242,45.606,158.930
C05035=1032.948,351.385,-131.847,172.236,45.605,158.929
C05036=1032.940,351.138,-131.810,172.230,45.603,158.928
C05037=1032.933,350.891,-131.771,172.223,45.601,158.927
C05038=1032.925,350.644,-131.734,172.218,45.599,158.926
C05039=1032.912,350.247,-131.673,172.207,45.596,158.924
C05040=1032.900,349.850,-131.613,172.197,45.593,158.922
C05041=1032.888,349.453,-131.552,172.188,45.591,158.920
C05042=1032.875,349.057,-131.491,172.178,45.588,158.919
C05043=1032.868,348.810,-131.454,172.173,45.586,158.917
C05044=1032.860,348.563,-131.417,172.166,45.584,158.916
C05045=1032.852,348.316,-131.379,172.160,45.583,158.915
C05046=1032.845,348.068,-131.341,172.155,45.581,158.914
C05047=1032.837,347.821,-131.304,172.148,45.579,158.913
C05048=1032.829,347.574,-131.267,172.142,45.578,158.912
C05049=1032.821,347.327,-131.230,172.136,45.576,158.911
C05050=1032.814,347.080,-131.192,172.130,45.574,158.910
C05051=1032.806,346.833,-131.156,172.124,45.572,158.909
C05052=1032.798,346.585,-131.118,172.118,45.571,158.908
C05053=1032.790,346.338,-131.081,172.113,45.569,158.907
C05054=1032.783,346.091,-131.043,172.106,45.567,158.906
C05055=1032.775,345.844,-131.006,172.101,45.566,158.905
C05056=1032.768,345.597,-130.969,172.095,45.564,158.904
C05057=1032.760,345.351,-130.932,172.089,45.563,158.903
C05058=1032.753,345.103,-130.894,172.083,45.561,158.902
C05059=1032.745,344.856,-130.857,172.077,45.560,158.901
C05060=1032.737,344.609,-130.820,172.071,45.558,158.900
C05061=1032.730,344.362,-130.783,172.066,45.556,158.899
C05062=1032.722,344.115,-130.746,172.059,45.554,158.898
C05063=1032.714,343.868,-130.709,172.054,45.553,158.897
C05064=1032.708,343.620,-130.672,172.048,45.552,158.896
C05065=1032.700,343.373,-130.635,172.041,45.550,158.895
C05066=1032.692,343.126,-130.598,172.036,45.548,158.894
C05067=1032.685,342.879,-130.562,172.030,45.547,158.893
C05068=1032.677,342.632,-130.524,172.025,45.545,158.892
C05069=1032.669,342.385,-130.487,172.019,45.544,158.891
C05070=1032.662,342.137,-130.450,172.014,45.542,158.890
C05071=1032.655,341.890,-130.413,172.007,45.541,158.889
C05072=1032.647,341.643,-130.377,172.002,45.539,158.888
C05073=1032.640,341.396,-130.340,171.996,45.538,158.887
C05074=1032.632,341.148,-130.303,171.990,45.537,158.886
C05075=1032.625,340.901,-130.266,171.985,45.535,158.885
C05076=1032.617,340.654,-130.230,171.978,45.533,158.884
C05077=1032.609,340.407,-130.193,171.973,45.532,158.883
C05078=1032.601,340.159,-130.157,171.967,45.531,158.882
C05079=1032.594,339.913,-130.121,171.962,45.529,158.881
C05080=1032.587,339.666,-130.083,171.956,45.528,158.880
C05081=1032.579,339.418,-130.047,171.951,45.526,158.879
C05082=1032.572,339.171,-130.011,171.945,45.525,158.879
C05083=1032.564,338.923,-129.975,171.939,45.524,158.878
C05084=1032.556,338.676,-129.938,171.933,45.523,158.877
C05085=1032.550,338.429,-129.901,171.928,45.521,158.876
C05086=1032.542,338.182,-129.865,171.922,45.520,158.875
C05087=1032.534,337.934,-129.829,171.917,45.518,158.874
C05088=1032.527,337.687,-129.793,171.911,45.517,158.873
C05089=1032.519,337.440,-129.756,171.906,45.516,158.872
C05090=1032.512,337.193,-129.720,171.900,45.514,158.871
C05091=1032.505,336.946,-129.683,171.895,45.514,158.870
C05092=1032.497,336.698,-129.647,171.890,45.512,158.870
C05093=1032.489,336.451,-129.611,171.883,45.511,158.869
C05094=1032.482,336.204,-129.575,171.878,45.509,158.868
C05095=1032.470,335.803,-129.516,171.869,45.508,158.866
C05096=1032.458,335.404,-129.457,171.860,45.506,158.865
C05097=1032.447,335.004,-129.399,171.851,45.503,158.863
C05098=1032.434,334.603,-129.341,171.842,45.501,158.862
C05099=1032.428,334.356,-129.304,171.837,45.500,158.861
C05100=1032.420,334.109,-129.269,171.831,45.499,158.860
C05101=1032.412,333.861,-129.233,171.826,45.497,158.859
C05102=1032.405,333.614,-129.197,171.821,45.496,158.859
C05103=1032.397,333.367,-129.161,171.815,45.495,158.858
C05104=1032.390,333.120,-129.126,171.810,45.494,158.857
C05105=1032.383,332.872,-129.090,171.804,45.493,158.856
C05106=1032.375,332.625,-129.053,171.799,45.492,158.855
C05107=1032.368,332.377,-129.018,171.794,45.491,158.854
C05108=1032.361,332.130,-128.982,171.788,45.489,158.853
C05109=1032.353,331.883,-128.946,171.783,45.489,158.853
C05110=1032.346,331.635,-128.911,171.777,45.487,158.852
C05111=1032.339,331.388,-128.875,171.772,45.486,158.851
C05112=1032.331,331.141,-128.839,171.767,45.485,158.850
C05113=1032.324,330.894,-128.804,171.761,45.484,158.849
C05114=1032.316,330.646,-128.768,171.756,45.483,158.848
C05115=1032.309,330.399,-128.733,171.751,45.482,158.848
C05116=1032.302,330.152,-128.696,171.745,45.481,158.847
C05117=1032.295,329.904,-128.661,171.740,45.480,158.846
C05118=1032.287,329.657,-128.625,171.735,45.478,158.845
C05119=1032.281,329.409,-128.590,171.731,45.477,158.844
C05120=1032.273,329.161,-128.554,171.725,45.477,158.844
C05121=1032.265,328.915,-128.519,171.720,45.475,158.843
C05122=1032.258,328.667,-128.484,171.715,45.474,158.842
C05123=1032.251,328.420,-128.448,171.709,45.474,158.841
C05124=1032.244,328.173,-128.413,171.704,45.472,158.840
C05125=1032.237,327.925,-128.377,171.699,45.471,158.840
C05126=1032.229,327.678,-128.343,171.693,45.471,158.839
C05127=1032.222,327.430,-128.306,171.688,45.470,158.838
C05128=1032.214,327.183,-128.272,171.683,45.469,158.837
C05129=1032.207,326.935,-128.236,171.678,45.467,158.836
C05130=1032.199,326.688,-128.202,171.672,45.467,158.836
C05131=1032.192,326.441,-128.167,171.668,45.466,158.835
C05132=1032.184,326.193,-128.132,171.663,45.465,158.834
C05133=1032.178,325.946,-128.097,171.657,45.464,158.834
C05134=1032.169,325.698,-128.062,171.652,45.463,158.833
C05135=1032.163,325.450,-128.027,171.647,45.463,158.832
C05136=1032.155,325.203,-127.992,171.642,45.462,158.831
C05137=1032.147,324.956,-127.957,171.636,45.461,158.831
C05138=1032.140,324.708,-127.922,171.632,45.460,158.830
C05139=1032.133,324.461,-127.888,171.627,45.459,158.829
C05140=1032.125,324.213,-127.852,171.622,45.458,158.828
C05141=1032.118,323.966,-127.817,171.616,45.458,158.828
C05142=1032.111,323.719,-127.782,171.611,45.457,158.827
C05143=1032.104,323.472,-127.748,171.606,45.456,158.826
C05144=1032.097,323.223,-127.713,171.602,45.455,158.825
C05145=1032.089,322.976,-127.678,171.596,45.454,158.825
C05146=1032.082,322.729,-127.644,171.591,45.453,158.824
C05147=1032.075,322.482,-127.609,171.586,45.453,158.823
C05148=1032.067,322.234,-127.574,171.581,45.452,158.823
C05149=1032.060,321.986,-127.539,171.576,45.451,158.822
C05150=1032.053,321.739,-127.505,171.571,45.450,158.821
C05151=1032.041,321.334,-127.448,171.562,45.449,158.820
C05152=1032.029,320.929,-127.391,171.555,45.448,158.819
C05153=1032.018,320.525,-127.335,171.547,45.446,158.818
C05154=1032.006,320.120,-127.278,171.538,45.445,158.817
C05155=1031.999,319.873,-127.243,171.534,45.445,158.816
C05156=1031.992,319.625,-127.209,171.529,45.444,158.815
C05157=1031.985,319.378,-127.174,171.524,45.443,158.815
C05158=1031.977,319.130,-127.139,171.518,45.443,158.814
C05159=1031.970,318.883,-127.106,171.513,45.442,158.813
C05160=1031.963,318.635,-127.070,171.509,45.441,158.812
C05161=1031.956,318.388,-127.037,171.504,45.441,158.812
C05162=1031.949,318.140,-127.002,171.499,45.440,158.811
C05163=1031.942,317.893,-126.968,171.494,45.439,158.810
C05164=1031.934,317.645,-126.933,171.490,45.438,158.810
C05165=1031.928,317.397,-126.899,171.485,45.438,158.809
C05166=1031.920,317.150,-126.864,171.480,45.437,158.808
C05167=1031.914,316.902,-126.830,171.474,45.436,158.808
C05168=1031.906,316.655,-126.795,171.470,45.436,158.807
C05169=1031.899,316.408,-126.761,171.465,45.435,158.806
C05170=1031.893,316.160,-126.727,171.460,45.435,158.806
C05171=1031.885,315.913,-126.692,171.455,45.434,158.805
C05172=1031.879,315.665,-126.658,171.451,45.433,158.804
C05173=1031.872,315.418,-126.625,171.446,45.432,158.804
C05174=1031.865,315.171,-126.590,171.441,45.432,158.803
C05175=1031.858,314.923,-126.556,171.437,45.431,158.802
C05176=1031.851,314.675,-126.522,171.432,45.430,158.802
C05177=1031.844,314.428,-126.487,171.427,45.429,158.801
C05178=1031.837,314.180,-126.453,171.422,45.429,158.800
C05179=1031.830,313.932,-126.419,171.418,45.428,158.800
C05180=1031.823,313.684,-126.385,171.413,45.428,158.799
C05181=1031.816,313.438,-126.350,171.408,45.427,158.798
C05182=1031.809,313.190,-126.317,171.404,45.427,158.798
C05183=1031.803,312.942,-126.282,171.399,45.426,158.797
C05184=1031.796,312.695,-126.248,171.394,45.425,158.797
C05185=1031.788,312.447,-126.215,171.389,45.425,158.796
C05186=1031.782,312.200,-126.180,171.385,45.424,158.795
C05187=1031.775,311.953,-126.146,171.380,45.423,158.795
C05188=1031.769,311.705,-126.112,171.375,45.423,158.794
C05189=1031.761,311.457,-126.078,171.370,45.422,158.793
C05190=1031.755,311.210,-126.044,171.366,45.422,158.793
C05191=1031.748,310.962,-126.010,171.361,45.422,158.792
C05192=1031.741,310.714,-125.977,171.357,45.421,158.792
C05193=1031.733,310.467,-125.944,171.351,45.421,158.791
C05194=1031.725,310.219,-125.910,171.346,45.420,158.790
C05195=1031.718,309.971,-125.876,171.342,45.420,158.790
C05196=1031.712,309.724,-125.843,171.337,45.420,158.789
C05197=1031.704,309.476,-125.810,171.333,45.419,158.789
C05198=1031.697,309.229,-125.777,171.328,45.419,158.788
C05199=1031.690,308.981,-125.743,171.323,45.419,158.788
C05200=1031.683,308.734,-125.709,171.319,45.419,158.787
C05201=1031.676,308.486,-125.676,171.314,45.418,158.787
C05202=1031.668,308.238,-125.643,171.309,45.417,158.786
C05203=1031.661,307.991,-125.609,171.305,45.417,158.785
C05204=1031.655,307.743,-125.576,171.300,45.417,158.785
C05205=1031.648,307.495,-125.543,171.296,45.416,158.784
C05206=1031.640,307.248,-125.509,171.291,45.416,158.784
C05207=1031.628,306.848,-125.456,171.284,45.416,158.783
C05208=1031.617,306.448,-125.402,171.276,45.415,158.782
C05209=1031.605,306.049,-125.349,171.269,45.414,158.781
C05210=1031.594,305.649,-125.295,171.262,45.414,158.780
C05211=1031.588,305.401,-125.262,171.258,45.414,158.780
C05212=1031.581,305.154,-125.228,171.253,45.413,158.779
C05213=1031.573,304.906,-125.196,171.249,45.413,158.778
C05214=1031.567,304.659,-125.162,171.244,45.413,158.778
C05215=1031.560,304.410,-125.129,171.240,45.412,158.777
C05216=1031.552,304.163,-125.095,171.235,45.412,158.777
C05217=1031.545,303.915,-125.063,171.230,45.412,158.776
C05218=1031.538,303.668,-125.029,171.226,45.412,158.776
C05219=1031.532,303.420,-124.997,171.222,45.412,158.775
C05220=1031.525,303.172,-124.964,171.217,45.412,158.775
C05221=1031.518,302.925,-124.931,171.212,45.411,158.774
C05222=1031.511,302.677,-124.898,171.208,45.411,158.774
C05223=1031.504,302.429,-124.865,171.203,45.411,158.773
C05224=1031.497,302.182,-124.832,171.200,45.410,158.773
C05225=1031.490,301.934,-124.799,171.195,45.410,158.772
C05226=1031.483,301.686,-124.766,171.191,45.410,158.772
C05227=1031.477,301.439,-124.733,171.186,45.410,158.771
C05228=1031.469,301.191,-124.700,171.182,45.410,158.771
C05229=1031.463,300.944,-124.667,171.177,45.409,158.770
C05230=1031.456,300.695,-124.634,171.173,45.409,158.769
C05231=1031.449,300.448,-124.602,171.168,45.409,158.769
C05232=1031.442,300.200,-124.568,171.165,45.409,158.769
C05233=1031.435,299.953,-124.535,171.160,45.408,158.768
C05234=1031.429,299.704,-124.502,171.156,45.408,158.767
C05235=1031.421,299.457,-124.470,171.151,45.408,158.767
C05236=1031.415,299.210,-124.437,171.147,45.408,158.767
C05237=1031.408,298.961,-124.404,171.142,45.408,158.766
C05238=1031.401,298.714,-124.372,171.138,45.407,158.765
C05239=1031.394,298.466,-124.339,171.134,45.407,158.765
C05240=1031.388,298.219,-124.305,171.130,45.407,158.765
C05241=1031.381,297.971,-124.273,171.125,45.407,158.764
C05242=1031.374,297.723,-124.240,171.121,45.407,158.763
C05243=1031.368,297.476,-124.207,171.116,45.406,158.763
C05244=1031.361,297.228,-124.175,171.113,45.406,158.763
C05245=1031.354,296.980,-124.142,171.108,45.406,158.762
C05246=1031.347,296.732,-124.109,171.103,45.406,158.761
C05247=1031.341,296.485,-124.077,171.099,45.406,158.761
C05248=1031.333,296.237,-124.044,171.095,45.406,158.761
C05249=1031.327,295.989,-124.011,171.091,45.405,158.760
C05250=1031.321,295.741,-123.979,171.087,45.406,158.760
C05251=1031.315,295.493,-123.947,171.082,45.405,158.759
C05252=1031.307,295.245,-123.914,171.078,45.406,158.759
C05253=1031.301,294.998,-123.881,171.073,45.405,158.758
C05254=1031.295,294.750,-123.849,171.070,45.405,158.758
C05255=1031.287,294.502,-123.816,171.065,45.405,158.757
C05256=1031.281,294.255,-123.783,171.061,45.405,158.757
C05257=1031.274,294.007,-123.752,171.057,45.405,158.756
C05258=1031.267,293.759,-123.720,171.053,45.404,158.756
C05259=1031.260,293.511,-123.687,171.049,45.405,158.755
C05260=1031.253,293.263,-123.655,171.044,45.404,158.755
C05261=1031.246,293.016,-123.623,171.040,45.405,158.755
C05262=1031.240,292.768,-123.590,171.035,45.405,158.754
C05263=1031.229,292.385,-123.541,171.030,45.404,158.753
C05264=1031.219,292.003,-123.491,171.023,45.405,158.753
C05265=1031.208,291.620,-123.442,171.016,45.405,158.752
C05266=1031.198,291.237,-123.392,171.010,45.405,158.751
C05267=1031.191,290.989,-123.361,171.006,45.405,158.751
C05268=1031.183,290.741,-123.328,171.002,45.405,158.751
C05269=1031.176,290.493,-123.297,170.998,45.405,158.750
C05270=1031.170,290.246,-123.264,170.993,45.405,158.750
C05271=1031.163,289.998,-123.233,170.989,45.406,158.749
C05272=1031.156,289.751,-123.200,170.985,45.405,158.749
C05273=1031.149,289.502,-123.169,170.981,45.405,158.749
C05274=1031.142,289.254,-123.137,170.977,45.406,158.748
C05275=1031.136,289.006,-123.104,170.973,45.406,158.748
C05276=1031.129,288.759,-123.073,170.969,45.405,158.747
C05277=1031.122,288.511,-123.041,170.965,45.406,158.747
C05278=1031.116,288.263,-123.009,170.960,45.406,158.746
C05279=1031.109,288.015,-122.978,170.956,45.406,158.746
C05280=1031.102,287.767,-122.946,170.953,45.406,158.746
C05281=1031.095,287.519,-122.913,170.948,45.406,158.745
C05282=1031.089,287.271,-122.882,170.944,45.406,158.745
C05283=1031.082,287.023,-122.851,170.940,45.407,158.744
C05284=1031.075,286.776,-122.818,170.936,45.407,158.744
C05285=1031.068,286.528,-122.787,170.932,45.407,158.744
C05286=1031.061,286.280,-122.756,170.927,45.407,158.743
C05287=1031.055,286.032,-122.724,170.924,45.407,158.743
C05288=1031.048,285.785,-122.693,170.920,45.407,158.742
C05289=1031.041,285.537,-122.661,170.916,45.407,158.742
C05290=1031.034,285.289,-122.630,170.911,45.408,158.742
C05291=1031.027,285.041,-122.597,170.908,45.408,158.741
C05292=1031.020,284.793,-122.566,170.904,45.408,158.741
C05293=1031.013,284.545,-122.535,170.899,45.408,158.741
C05294=1031.007,284.297,-122.503,170.896,45.409,158.740
C05295=1031.000,284.049,-122.472,170.892,45.409,158.740
C05296=1030.993,283.801,-122.440,170.887,45.409,158.739
C05297=1030.986,283.553,-122.409,170.884,45.409,158.739
C05298=1030.980,283.305,-122.377,170.880,45.410,158.739
C05299=1030.972,283.058,-122.347,170.875,45.410,158.738
C05300=1030.966,282.810,-122.315,170.871,45.410,158.738
C05301=1030.959,282.562,-122.284,170.868,45.410,158.738
C05302=1030.952,282.314,-122.253,170.864,45.411,158.737
C05303=1030.946,282.066,-122.221,170.859,45.411,158.737
C05304=1030.939,281.818,-122.190,170.856,45.411,158.737
C05305=1030.932,281.570,-122.159,170.852,45.411,158.736
C05306=1030.925,281.322,-122.127,170.847,45.412,158.736
C05307=1030.919,281.074,-122.096,170.844,45.412,158.736
C05308=1030.912,280.826,-122.064,170.840,45.413,158.735
C05309=1030.905,280.578,-122.033,170.837,45.413,158.735
C05310=1030.899,280.330,-122.002,170.832,45.413,158.735
C05311=1030.891,280.082,-121.971,170.828,45.413,158.734
C05312=1030.885,279.834,-121.940,170.825,45.413,158.734
C05313=1030.879,279.587,-121.909,170.821,45.414,158.733
C05314=1030.872,279.339,-121.877,170.816,45.414,158.733
C05315=1030.865,279.091,-121.847,170.813,45.414,158.733
C05316=1030.859,278.843,-121.815,170.809,45.415,158.732
C05317=1030.852,278.595,-121.784,170.806,45.415,158.732
C05318=1030.845,278.347,-121.752,170.801,45.415,158.732
C05319=1030.835,277.976,-121.707,170.796,45.416,158.731
C05320=1030.825,277.605,-121.660,170.789,45.416,158.731
C05321=1030.815,277.235,-121.614,170.784,45.417,158.730
C05322=1030.805,276.864,-121.568,170.778,45.417,158.730
C05323=1030.798,276.616,-121.537,170.775,45.418,158.730
C05324=1030.791,276.368,-121.506,170.770,45.418,158.729
C05325=1030.784,276.120,-121.475,170.766,45.419,158.729
C05326=1030.779,275.872,-121.445,170.763,45.419,158.728
C05327=1030.771,275.625,-121.414,170.759,45.420,158.728
C05328=1030.765,275.376,-121.383,170.755,45.420,158.728
C05329=1030.758,275.128,-121.352,170.751,45.420,158.728
C05330=1030.751,274.880,-121.322,170.747,45.421,158.727
C05331=1030.744,274.632,-121.290,170.744,45.421,158.727
C05332=1030.738,274.385,-121.260,170.739,45.421,158.727
C05333=1030.731,274.136,-121.230,170.736,45.422,158.726
C05334=1030.724,273.888,-121.198,170.732,45.422,158.726
C05335=1030.718,273.640,-121.168,170.729,45.422,158.726
C05336=1030.710,273.392,-121.137,170.725,45.423,158.725
C05337=1030.705,273.144,-121.106,170.720,45.424,158.725
C05338=1030.697,272.896,-121.076,170.717,45.424,158.725
C05339=1030.691,272.648,-121.045,170.713,45.425,158.725
C05340=1030.684,272.400,-121.015,170.710,45.425,158.724
C05341=1030.678,272.152,-120.984,170.706,45.426,158.724
C05342=1030.671,271.904,-120.953,170.702,45.426,158.724
C05343=1030.664,271.656,-120.923,170.698,45.427,158.723
C05344=1030.657,271.408,-120.892,170.694,45.427,158.723
C05345=1030.651,271.160,-120.862,170.691,45.428,158.723
C05346=1030.644,270.912,-120.831,170.687,45.428,158.723
C05347=1030.637,270.664,-120.801,170.684,45.429,158.722
C05348=1030.631,270.416,-120.770,170.679,45.429,158.722
C05349=1030.624,270.168,-120.740,170.676,45.430,158.722
C05350=1030.618,269.919,-120.710,170.672,45.430,158.721
C05351=1030.610,269.671,-120.679,170.669,45.431,158.721
C05352=1030.604,269.424,-120.649,170.665,45.431,158.721
C05353=1030.597,269.176,-120.618,170.661,45.432,158.721
C05354=1030.590,268.928,-120.588,170.657,45.432,158.720
C05355=1030.584,268.680,-120.558,170.653,45.433,158.720
C05356=1030.577,268.432,-120.528,170.650,45.434,158.720
C05357=1030.570,268.183,-120.497,170.646,45.434,158.720
C05358=1030.564,267.936,-120.467,170.643,45.435,158.719
C05359=1030.557,267.687,-120.437,170.639,45.435,158.719
C05360=1030.551,267.439,-120.406,170.636,45.436,158.719
C05361=1030.544,267.191,-120.377,170.632,45.437,158.719
C05362=1030.537,266.943,-120.346,170.628,45.437,158.718
C05363=1030.530,266.695,-120.316,170.624,45.438,158.718
C05364=1030.524,266.447,-120.286,170.621,45.438,158.718
C05365=1030.517,266.199,-120.256,170.617,45.439,158.717
C05366=1030.510,265.951,-120.226,170.614,45.439,158.717
C05367=1030.504,265.703,-120.195,170.610,45.440,158.717
C05368=1030.497,265.454,-120.166,170.607,45.440,158.717
C05369=1030.490,265.206,-120.136,170.603,45.441,158.717
C05370=1030.483,264.958,-120.106,170.599,45.442,158.716
C05371=1030.477,264.710,-120.076,170.595,45.442,158.716
C05372=1030.470,264.462,-120.046,170.592,45.443,158.716
C05373=1030.463,264.214,-120.015,170.588,45.444,158.716
C05374=1030.457,263.966,-119.986,170.585,45.444,158.715
C05375=1030.447,263.599,-119.942,170.579,45.445,158.715
C05376=1030.437,263.234,-119.898,170.574,45.447,158.715
C05377=1030.427,262.868,-119.854,170.568,45.447,158.714
C05378=1030.418,262.502,-119.809,170.563,45.448,158.714
C05379=1030.411,262.254,-119.779,170.560,45.449,158.714
C05380=1030.404,262.006,-119.749,170.556,45.450,158.714
C05381=1030.398,261.757,-119.720,170.553,45.450,158.713
C05382=1030.391,261.510,-119.690,170.549,45.451,158.713
C05383=1030.385,261.261,-119.660,170.546,45.452,158.713
